Yaskawa INFORM job: A_ROOF_SIDE_0617_2_PAINT_1.JBI

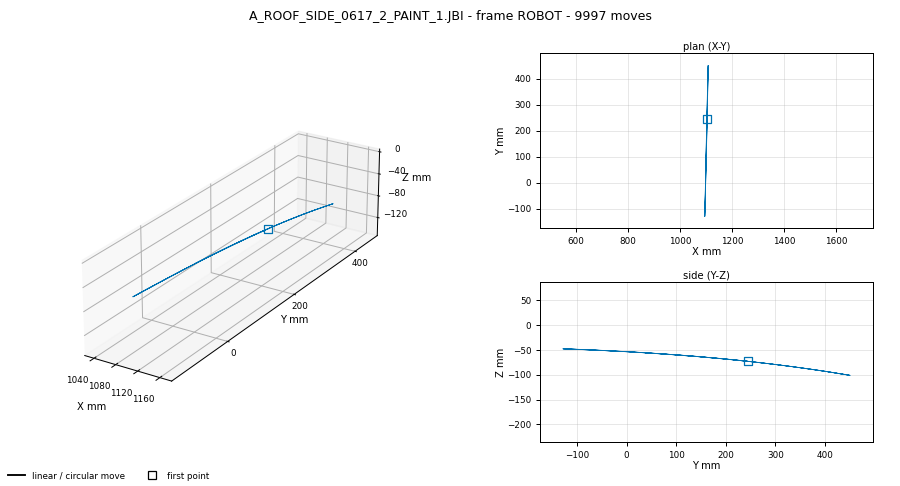
[picture p0: tool path of A_ROOF_SIDE_0617_2_PAINT_1.JBI in frame ROBOT, 9997 of 9997 moves have a stored position in this frame; points joined in program order, loops and branches not executed]
/JOB
//NAME A_ROOF_SIDE_0617_2_PAINT1
//POS
///NPOS 9997,0,0,0,0,0
///TOOL 1
///USER 0
///POSTYPE ROBOT
///RECTAN
///RCONF 1,0,0,0,0,0,0,0,0,0,0,0,0,0,0,0,0,0,0,0,0,0,0,0
C00000=1104.721,243.899,-72.511,179.198,14.617,151.233
C00001=1104.715,243.651,-72.485,179.194,14.617,151.234
C00002=1104.709,243.403,-72.458,179.190,14.617,151.234
C00003=1104.703,243.154,-72.431,179.186,14.617,151.235
C00004=1104.698,242.906,-72.404,179.183,14.617,151.236
C00005=1104.693,242.657,-72.378,179.179,14.617,151.237
C00006=1104.687,242.408,-72.352,179.175,14.617,151.238
C00007=1104.681,242.160,-72.325,179.171,14.616,151.238
C00008=1104.676,241.912,-72.298,179.167,14.617,151.239
C00009=1104.670,241.663,-72.272,179.163,14.616,151.240
C00010=1104.664,241.414,-72.246,179.159,14.616,151.241
C00011=1104.659,241.166,-72.219,179.155,14.616,151.242
C00012=1104.653,240.918,-72.192,179.151,14.616,151.243
C00013=1104.647,240.669,-72.166,179.148,14.616,151.244
C00014=1104.641,240.420,-72.140,179.144,14.616,151.244
C00015=1104.636,240.172,-72.113,179.140,14.616,151.245
C00016=1104.630,239.924,-72.086,179.136,14.616,151.246
C00017=1104.624,239.675,-72.060,179.132,14.616,151.247
C00018=1104.619,239.426,-72.034,179.129,14.616,151.248
C00019=1104.613,239.178,-72.007,179.125,14.616,151.249
C00020=1104.607,238.929,-71.981,179.121,14.616,151.250
C00021=1104.602,238.680,-71.955,179.117,14.616,151.250
C00022=1104.596,238.432,-71.928,179.113,14.616,151.251
C00023=1104.590,238.183,-71.902,179.110,14.616,151.252
C00024=1104.585,237.935,-71.875,179.105,14.615,151.253
C00025=1104.579,237.686,-71.849,179.101,14.615,151.254
C00026=1104.573,237.437,-71.823,179.097,14.615,151.254
C00027=1104.568,237.189,-71.796,179.094,14.615,151.255
C00028=1104.562,236.940,-71.770,179.090,14.615,151.256
C00029=1104.554,236.578,-71.732,179.084,14.615,151.257
C00030=1104.545,236.215,-71.694,179.078,14.615,151.259
C00031=1104.538,235.854,-71.656,179.073,14.615,151.260
C00032=1104.529,235.491,-71.618,179.067,14.615,151.261
C00033=1104.524,235.243,-71.591,179.063,14.615,151.262
C00034=1104.518,234.994,-71.565,179.059,14.615,151.263
C00035=1104.512,234.745,-71.538,179.056,14.615,151.264
C00036=1104.507,234.496,-71.513,179.052,14.615,151.264
C00037=1104.500,234.248,-71.486,179.048,14.615,151.265
C00038=1104.495,233.999,-71.461,179.044,14.615,151.266
C00039=1104.490,233.751,-71.435,179.040,14.615,151.267
C00040=1104.484,233.503,-71.408,179.037,14.615,151.268
C00041=1104.479,233.254,-71.382,179.033,14.615,151.269
C00042=1104.473,233.005,-71.357,179.029,14.615,151.270
C00043=1104.467,232.757,-71.330,179.025,14.615,151.270
C00044=1104.461,232.508,-71.304,179.021,14.615,151.271
C00045=1104.456,232.259,-71.279,179.017,14.615,151.272
C00046=1104.450,232.011,-71.253,179.014,14.615,151.273
C00047=1104.444,231.762,-71.227,179.010,14.615,151.274
C00048=1104.439,231.513,-71.201,179.006,14.615,151.275
C00049=1104.433,231.265,-71.174,179.002,14.615,151.276
C00050=1104.427,231.016,-71.149,178.998,14.615,151.276
C00051=1104.422,230.767,-71.123,178.994,14.615,151.277
C00052=1104.417,230.519,-71.098,178.991,14.616,151.278
C00053=1104.411,230.271,-71.071,178.987,14.616,151.279
C00054=1104.405,230.022,-71.046,178.983,14.615,151.280
C00055=1104.399,229.773,-71.020,178.979,14.615,151.281
C00056=1104.393,229.524,-70.994,178.975,14.616,151.282
C00057=1104.388,229.275,-70.968,178.972,14.616,151.282
C00058=1104.383,229.027,-70.943,178.968,14.616,151.283
C00059=1104.376,228.779,-70.917,178.964,14.616,151.284
C00060=1104.371,228.530,-70.891,178.960,14.616,151.285
C00061=1104.365,228.282,-70.865,178.956,14.616,151.286
C00062=1104.359,228.033,-70.840,178.952,14.616,151.287
C00063=1104.354,227.784,-70.814,178.948,14.616,151.288
C00064=1104.348,227.536,-70.789,178.944,14.616,151.289
C00065=1104.342,227.287,-70.763,178.941,14.617,151.290
C00066=1104.336,227.038,-70.737,178.937,14.617,151.290
C00067=1104.331,226.789,-70.711,178.933,14.616,151.291
C00068=1104.325,226.541,-70.686,178.929,14.616,151.292
C00069=1104.320,226.292,-70.661,178.925,14.617,151.293
C00070=1104.314,226.043,-70.635,178.921,14.617,151.294
C00071=1104.309,225.795,-70.610,178.918,14.617,151.295
C00072=1104.302,225.546,-70.584,178.914,14.617,151.296
C00073=1104.297,225.297,-70.558,178.910,14.617,151.296
C00074=1104.291,225.049,-70.533,178.906,14.617,151.297
C00075=1104.286,224.800,-70.507,178.902,14.617,151.298
C00076=1104.280,224.552,-70.482,178.898,14.617,151.299
C00077=1104.274,224.303,-70.456,178.894,14.617,151.300
C00078=1104.269,224.055,-70.431,178.891,14.617,151.301
C00079=1104.263,223.806,-70.405,178.887,14.617,151.302
C00080=1104.257,223.557,-70.380,178.883,14.617,151.302
C00081=1104.249,223.186,-70.342,178.877,14.618,151.304
C00082=1104.241,222.816,-70.304,178.871,14.618,151.305
C00083=1104.232,222.445,-70.267,178.866,14.618,151.306
C00084=1104.224,222.074,-70.228,178.860,14.619,151.308
C00085=1104.218,221.826,-70.203,178.857,14.619,151.309
C00086=1104.212,221.577,-70.179,178.853,14.619,151.310
C00087=1104.207,221.328,-70.153,178.849,14.619,151.310
C00088=1104.201,221.079,-70.127,178.845,14.619,151.311
C00089=1104.195,220.831,-70.102,178.841,14.619,151.312
C00090=1104.190,220.582,-70.077,178.837,14.620,151.313
C00091=1104.184,220.334,-70.052,178.833,14.620,151.314
C00092=1104.178,220.085,-70.027,178.829,14.620,151.315
C00093=1104.172,219.836,-70.002,178.826,14.620,151.316
C00094=1104.167,219.587,-69.977,178.822,14.620,151.317
C00095=1104.161,219.339,-69.951,178.818,14.620,151.317
C00096=1104.155,219.090,-69.926,178.814,14.620,151.318
C00097=1104.150,218.841,-69.901,178.810,14.620,151.319
C00098=1104.144,218.593,-69.876,178.806,14.620,151.320
C00099=1104.139,218.345,-69.851,178.803,14.620,151.321
C00100=1104.133,218.095,-69.826,178.799,14.620,151.322
C00101=1104.127,217.846,-69.800,178.796,14.621,151.323
C00102=1104.122,217.598,-69.776,178.792,14.621,151.324
C00103=1104.116,217.349,-69.751,178.788,14.621,151.324
C00104=1104.110,217.101,-69.726,178.784,14.622,151.325
C00105=1104.104,216.852,-69.701,178.780,14.622,151.326
C00106=1104.099,216.603,-69.676,178.776,14.622,151.327
C00107=1104.093,216.354,-69.651,178.772,14.622,151.328
C00108=1104.087,216.106,-69.626,178.768,14.622,151.329
C00109=1104.082,215.857,-69.601,178.764,14.622,151.330
C00110=1104.076,215.608,-69.576,178.761,14.622,151.331
C00111=1104.071,215.359,-69.551,178.757,14.623,151.332
C00112=1104.065,215.111,-69.526,178.753,14.623,151.332
C00113=1104.060,214.862,-69.502,178.749,14.623,151.333
C00114=1104.053,214.613,-69.476,178.745,14.623,151.334
C00115=1104.048,214.365,-69.452,178.742,14.624,151.335
C00116=1104.042,214.116,-69.427,178.738,14.624,151.336
C00117=1104.037,213.868,-69.402,178.734,14.624,151.337
C00118=1104.032,213.618,-69.377,178.730,14.624,151.338
C00119=1104.026,213.370,-69.352,178.726,14.624,151.339
C00120=1104.020,213.121,-69.328,178.723,14.624,151.340
C00121=1104.015,212.872,-69.303,178.719,14.625,151.340
C00122=1104.008,212.623,-69.278,178.715,14.625,151.341
C00123=1104.003,212.375,-69.254,178.711,14.625,151.342
C00124=1103.997,212.126,-69.229,178.707,14.625,151.343
C00125=1103.992,211.878,-69.204,178.703,14.625,151.344
C00126=1103.986,211.629,-69.180,178.699,14.625,151.345
C00127=1103.980,211.380,-69.155,178.696,14.626,151.346
C00128=1103.975,211.132,-69.130,178.692,14.626,151.347
C00129=1103.969,210.882,-69.106,178.688,14.626,151.348
C00130=1103.964,210.634,-69.081,178.684,14.627,151.348
C00131=1103.958,210.385,-69.057,178.681,14.627,151.349
C00132=1103.952,210.137,-69.032,178.677,14.627,151.350
C00133=1103.943,209.769,-68.996,178.671,14.628,151.352
C00134=1103.935,209.402,-68.960,178.666,14.628,151.353
C00135=1103.927,209.035,-68.923,178.660,14.628,151.354
C00136=1103.918,208.667,-68.887,178.654,14.628,151.356
C00137=1103.896,207.669,-68.790,178.625,14.626,151.361
C00138=1103.890,207.420,-68.765,178.621,14.626,151.362
C00139=1103.884,207.171,-68.741,178.617,14.628,151.364
C00140=1103.878,206.922,-68.717,178.613,14.628,151.365
C00141=1103.873,206.673,-68.692,178.609,14.630,151.366
C00142=1103.867,206.425,-68.669,178.605,14.631,151.367
C00143=1103.861,206.176,-68.644,178.600,14.632,151.368
C00144=1103.856,205.927,-68.620,178.597,14.633,151.369
C00145=1103.851,205.679,-68.596,178.592,14.634,151.370
C00146=1103.844,205.430,-68.572,178.589,14.635,151.372
C00147=1103.839,205.181,-68.547,178.584,14.636,151.373
C00148=1103.833,204.932,-68.523,178.580,14.637,151.374
C00149=1103.827,204.683,-68.498,178.576,14.638,151.375
C00150=1103.821,204.435,-68.475,178.572,14.639,151.376
C00151=1103.816,204.186,-68.450,178.568,14.640,151.377
C00152=1103.810,203.936,-68.427,178.564,14.641,151.378
C00153=1103.804,203.688,-68.403,178.560,14.642,151.379
C00154=1103.799,203.439,-68.379,178.556,14.643,151.381
C00155=1103.794,203.191,-68.354,178.552,14.644,151.382
C00156=1103.788,202.942,-68.330,178.547,14.645,151.383
C00157=1103.782,202.693,-68.306,178.544,14.646,151.384
C00158=1103.777,202.445,-68.282,178.539,14.647,151.385
C00159=1103.770,202.195,-68.259,178.536,14.648,151.386
C00160=1103.765,201.946,-68.234,178.531,14.649,151.387
C00161=1103.759,201.698,-68.211,178.527,14.650,151.388
C00162=1103.753,201.449,-68.186,178.524,14.651,151.389
C00163=1103.747,201.201,-68.162,178.519,14.652,151.391
C00164=1103.742,200.951,-68.139,178.516,14.654,151.392
C00165=1103.736,200.703,-68.115,178.511,14.655,151.393
C00166=1103.730,200.454,-68.091,178.508,14.656,151.394
C00167=1103.724,200.206,-68.067,178.503,14.657,151.395
C00168=1103.719,199.956,-68.043,178.499,14.658,151.396
C00169=1103.712,199.707,-68.019,178.495,14.659,151.397
C00170=1103.707,199.459,-67.995,178.491,14.660,151.399
C00171=1103.701,199.210,-67.972,178.487,14.661,151.400
C00172=1103.696,198.961,-67.948,178.483,14.662,151.401
C00173=1103.689,198.712,-67.924,178.479,14.663,151.402
C00174=1103.684,198.463,-67.900,178.475,14.664,151.403
C00175=1103.678,198.215,-67.877,178.471,14.665,151.404
C00176=1103.672,197.967,-67.853,178.467,14.666,151.405
C00177=1103.667,197.717,-67.829,178.463,14.667,151.406
C00178=1103.661,197.468,-67.805,178.459,14.668,151.407
C00179=1103.656,197.219,-67.782,178.455,14.669,151.409
C00180=1103.650,196.971,-67.758,178.451,14.670,151.410
C00181=1103.644,196.722,-67.734,178.447,14.671,151.411
C00182=1103.638,196.473,-67.711,178.443,14.672,151.412
C00183=1103.632,196.224,-67.687,178.439,14.672,151.413
C00184=1103.627,195.975,-67.663,178.435,14.674,151.414
C00185=1103.621,195.727,-67.640,178.431,14.675,151.415
C00186=1103.616,195.478,-67.616,178.427,14.676,151.416
C00187=1103.610,195.230,-67.593,178.423,14.677,151.417
C00188=1103.604,194.981,-67.570,178.419,14.677,151.418
C00189=1103.598,194.731,-67.545,178.415,14.679,151.420
C00190=1103.593,194.482,-67.522,178.411,14.680,151.421
C00191=1103.587,194.234,-67.498,178.407,14.681,151.422
C00192=1103.582,193.985,-67.475,178.403,14.681,151.423
C00193=1103.576,193.736,-67.452,178.399,14.682,151.424
C00194=1103.570,193.488,-67.428,178.396,14.683,151.425
C00195=1103.565,193.239,-67.405,178.391,14.684,151.426
C00196=1103.559,192.990,-67.381,178.387,14.686,151.427
C00197=1103.552,192.741,-67.358,178.383,14.686,151.428
C00198=1103.547,192.469,-67.332,178.379,14.687,151.429
C00199=1103.541,192.198,-67.307,178.375,14.688,151.431
C00200=1103.535,191.926,-67.281,178.371,14.690,151.432
C00201=1103.528,191.655,-67.255,178.366,14.690,151.433
C00202=1103.523,191.406,-67.232,178.362,14.691,151.434
C00203=1103.518,191.156,-67.209,178.358,14.693,151.435
C00204=1103.511,190.907,-67.185,178.354,14.693,151.436
C00205=1103.505,190.659,-67.162,178.350,14.694,151.437
C00206=1103.500,190.409,-67.138,178.347,14.695,151.438
C00207=1103.495,190.160,-67.115,178.342,14.696,151.439
C00208=1103.489,189.912,-67.092,178.339,14.697,151.440
C00209=1103.483,189.663,-67.069,178.335,14.698,151.442
C00210=1103.478,189.414,-67.045,178.330,14.699,151.443
C00211=1103.472,189.165,-67.022,178.327,14.700,151.444
C00212=1103.466,188.916,-66.999,178.323,14.700,151.445
C00213=1103.460,188.668,-66.976,178.319,14.702,151.446
C00214=1103.455,188.419,-66.952,178.315,14.702,151.447
C00215=1103.450,188.170,-66.929,178.312,14.704,151.448
C00216=1103.444,187.921,-66.906,178.307,14.704,151.449
C00217=1103.438,187.672,-66.883,178.303,14.705,151.450
C00218=1103.432,187.423,-66.860,178.300,14.706,151.451
C00219=1103.427,187.174,-66.837,178.296,14.706,151.452
C00220=1103.422,186.926,-66.814,178.292,14.708,151.453
C00221=1103.416,186.677,-66.791,178.288,14.708,151.454
C00222=1103.410,186.429,-66.768,178.284,14.709,151.455
C00223=1103.405,186.180,-66.745,178.280,14.710,151.456
C00224=1103.400,185.930,-66.721,178.276,14.711,151.457
C00225=1103.394,185.682,-66.698,178.273,14.712,151.458
C00226=1103.388,185.433,-66.675,178.269,14.713,151.459
C00227=1103.383,185.184,-66.652,178.265,14.713,151.460
C00228=1103.377,184.935,-66.629,178.261,14.714,151.461
C00229=1103.371,184.686,-66.607,178.257,14.716,151.463
C00230=1103.365,184.437,-66.584,178.253,14.717,151.464
C00231=1103.360,184.188,-66.561,178.249,14.718,151.465
C00232=1103.354,183.939,-66.538,178.245,14.719,151.466
C00233=1103.348,183.690,-66.515,178.241,14.719,151.467
C00234=1103.342,183.442,-66.492,178.237,14.720,151.468
C00235=1103.336,183.193,-66.469,178.234,14.721,151.469
C00236=1103.330,182.944,-66.446,178.230,14.722,151.470
C00237=1103.325,182.695,-66.424,178.226,14.723,151.471
C00238=1103.319,182.446,-66.401,178.222,14.724,151.472
C00239=1103.313,182.197,-66.378,178.219,14.725,151.473
C00240=1103.308,181.948,-66.355,178.214,14.726,151.474
C00241=1103.301,181.699,-66.333,178.211,14.727,151.475
C00242=1103.295,181.450,-66.310,178.207,14.728,151.476
C00243=1103.290,181.201,-66.287,178.202,14.728,151.477
C00244=1103.284,180.953,-66.264,178.199,14.730,151.478
C00245=1103.278,180.704,-66.241,178.195,14.730,151.479
C00246=1103.273,180.455,-66.218,178.191,14.732,151.481
C00247=1103.267,180.205,-66.196,178.187,14.732,151.481
C00248=1103.261,179.957,-66.174,178.184,14.733,151.482
C00249=1103.256,179.708,-66.151,178.180,14.734,151.484
C00250=1103.250,179.460,-66.128,178.175,14.734,151.485
C00251=1103.244,179.211,-66.105,178.172,14.736,151.486
C00252=1103.239,178.961,-66.083,178.168,14.736,151.487
C00253=1103.232,178.713,-66.061,178.165,14.737,151.488
C00254=1103.226,178.464,-66.038,178.160,14.738,151.489
C00255=1103.221,178.214,-66.016,178.157,14.739,151.490
C00256=1103.215,177.965,-65.993,178.153,14.740,151.491
C00257=1103.209,177.717,-65.971,178.149,14.741,151.492
C00258=1103.204,177.468,-65.948,178.145,14.742,151.493
C00259=1103.198,177.219,-65.925,178.141,14.742,151.494
C00260=1103.193,176.970,-65.902,178.138,14.744,151.495
C00261=1103.186,176.721,-65.880,178.133,14.744,151.496
C00262=1103.180,176.449,-65.856,178.129,14.745,151.497
C00263=1103.174,176.177,-65.831,178.126,14.746,151.498
C00264=1103.168,175.905,-65.807,178.122,14.747,151.499
C00265=1103.162,175.633,-65.782,178.117,14.748,151.500
C00266=1103.156,175.384,-65.760,178.113,14.748,151.501
C00267=1103.150,175.135,-65.737,178.110,14.750,151.502
C00268=1103.144,174.886,-65.715,178.106,14.750,151.503
C00269=1103.139,174.637,-65.692,178.102,14.751,151.504
C00270=1103.134,174.388,-65.670,178.098,14.752,151.505
C00271=1103.127,174.140,-65.648,178.095,14.753,151.506
C00272=1103.122,173.890,-65.626,178.091,14.753,151.507
C00273=1103.116,173.641,-65.603,178.086,14.754,151.509
C00274=1103.111,173.393,-65.581,178.083,14.755,151.509
C00275=1103.105,173.144,-65.559,178.079,14.756,151.510
C00276=1103.100,172.894,-65.536,178.076,14.757,151.511
C00277=1103.093,172.646,-65.514,178.072,14.757,151.512
C00278=1103.088,172.397,-65.492,178.068,14.759,151.513
C00279=1103.082,172.148,-65.469,178.064,14.759,151.514
C00280=1103.076,171.899,-65.448,178.061,14.760,151.515
C00281=1103.071,171.650,-65.425,178.057,14.760,151.516
C00282=1103.065,171.401,-65.403,178.053,14.761,151.517
C00283=1103.060,171.152,-65.381,178.050,14.762,151.518
C00284=1103.054,170.903,-65.358,178.045,14.763,151.519
C00285=1103.048,170.654,-65.337,178.042,14.764,151.520
C00286=1103.043,170.405,-65.314,178.038,14.764,151.521
C00287=1103.037,170.156,-65.292,178.035,14.765,151.522
C00288=1103.032,169.907,-65.270,178.031,14.766,151.523
C00289=1103.026,169.659,-65.247,178.027,14.766,151.524
C00290=1103.020,169.409,-65.226,178.023,14.767,151.525
C00291=1103.015,169.161,-65.204,178.019,14.768,151.526
C00292=1103.009,168.911,-65.182,178.016,14.769,151.527
C00293=1103.003,168.662,-65.159,178.012,14.769,151.528
C00294=1102.998,168.414,-65.138,178.009,14.770,151.529
C00295=1102.992,168.164,-65.116,178.005,14.771,151.530
C00296=1102.987,167.915,-65.094,178.002,14.772,151.531
C00297=1102.981,167.667,-65.072,177.997,14.772,151.532
C00298=1102.975,167.417,-65.049,177.993,14.773,151.533
C00299=1102.970,167.169,-65.028,177.990,14.774,151.534
C00300=1102.964,166.919,-65.006,177.986,14.774,151.535
C00301=1102.959,166.671,-64.983,177.983,14.775,151.536
C00302=1102.953,166.422,-64.962,177.979,14.776,151.537
C00303=1102.948,166.173,-64.940,177.976,14.777,151.538
C00304=1102.942,165.924,-64.918,177.972,14.777,151.539
C00305=1102.937,165.675,-64.896,177.969,14.778,151.540
C00306=1102.931,165.426,-64.875,177.964,14.779,151.541
C00307=1102.926,165.176,-64.853,177.960,14.779,151.542
C00308=1102.919,164.928,-64.830,177.957,14.780,151.542
C00309=1102.914,164.679,-64.808,177.953,14.780,151.543
C00310=1102.908,164.430,-64.787,177.950,14.782,151.544
C00311=1102.903,164.181,-64.765,177.946,14.782,151.545
C00312=1102.897,163.932,-64.743,177.943,14.783,151.546
C00313=1102.892,163.683,-64.721,177.939,14.783,151.547
C00314=1102.886,163.434,-64.700,177.935,14.784,151.548
C00315=1102.881,163.185,-64.678,177.932,14.785,151.549
C00316=1102.875,162.936,-64.656,177.928,14.785,151.550
C00317=1102.870,162.687,-64.635,177.925,14.786,151.551
C00318=1102.864,162.438,-64.613,177.921,14.786,151.552
C00319=1102.859,162.189,-64.591,177.917,14.787,151.553
C00320=1102.853,161.940,-64.569,177.913,14.788,151.554
C00321=1102.848,161.691,-64.548,177.910,14.789,151.555
C00322=1102.842,161.442,-64.526,177.906,14.789,151.556
C00323=1102.837,161.193,-64.504,177.902,14.789,151.557
C00324=1102.831,160.944,-64.483,177.899,14.791,151.558
C00325=1102.824,160.695,-64.461,177.895,14.791,151.559
C00326=1102.819,160.423,-64.437,177.892,14.792,151.560
C00327=1102.813,160.150,-64.415,177.888,14.792,151.560
C00328=1102.806,159.878,-64.391,177.883,14.793,151.562
C00329=1102.800,159.605,-64.367,177.879,14.794,151.563
C00330=1102.794,159.356,-64.346,177.876,14.795,151.564
C00331=1102.788,159.107,-64.324,177.872,14.795,151.564
C00332=1102.783,158.858,-64.302,177.869,14.796,151.565
C00333=1102.777,158.609,-64.281,177.865,14.797,151.566
C00334=1102.772,158.360,-64.260,177.862,14.798,151.567
C00335=1102.766,158.111,-64.238,177.858,14.798,151.568
C00336=1102.760,157.862,-64.217,177.854,14.798,151.569
C00337=1102.754,157.613,-64.195,177.851,14.799,151.570
C00338=1102.749,157.364,-64.174,177.847,14.799,151.571
C00339=1102.743,157.115,-64.153,177.844,14.800,151.572
C00340=1102.738,156.866,-64.131,177.840,14.801,151.573
C00341=1102.732,156.617,-64.110,177.836,14.802,151.574
C00342=1102.726,156.368,-64.089,177.832,14.802,151.575
C00343=1102.721,156.119,-64.068,177.829,14.803,151.576
C00344=1102.715,155.870,-64.046,177.825,14.804,151.577
C00345=1102.710,155.621,-64.024,177.822,14.804,151.577
C00346=1102.704,155.371,-64.004,177.818,14.805,151.578
C00347=1102.698,155.123,-63.982,177.815,14.806,151.579
C00348=1102.692,154.874,-63.961,177.811,14.806,151.580
C00349=1102.687,154.625,-63.939,177.807,14.806,151.581
C00350=1102.681,154.375,-63.918,177.804,14.807,151.582
C00351=1102.675,154.127,-63.897,177.800,14.807,151.583
C00352=1102.670,153.878,-63.877,177.797,14.808,151.584
C00353=1102.664,153.628,-63.855,177.793,14.809,151.585
C00354=1102.658,153.380,-63.834,177.790,14.810,151.586
C00355=1102.652,153.130,-63.813,177.786,14.810,151.586
C00356=1102.647,152.882,-63.792,177.783,14.811,151.587
C00357=1102.641,152.633,-63.770,177.779,14.811,151.588
C00358=1102.635,152.383,-63.749,177.776,14.812,151.589
C00359=1102.630,152.135,-63.728,177.772,14.812,151.590
C00360=1102.624,151.885,-63.707,177.769,14.813,151.591
C00361=1102.618,151.636,-63.686,177.765,14.814,151.592
C00362=1102.613,151.387,-63.665,177.761,14.814,151.593
C00363=1102.607,151.138,-63.644,177.758,14.815,151.594
C00364=1102.602,150.889,-63.623,177.754,14.815,151.595
C00365=1102.596,150.641,-63.602,177.751,14.816,151.596
C00366=1102.590,150.391,-63.581,177.747,14.816,151.596
C00367=1102.585,150.142,-63.560,177.744,14.817,151.597
C00368=1102.579,149.893,-63.539,177.740,14.817,151.598
C00369=1102.573,149.644,-63.517,177.737,14.818,151.599
C00370=1102.568,149.395,-63.497,177.733,14.818,151.600
C00371=1102.562,149.146,-63.476,177.730,14.819,151.601
C00372=1102.557,148.896,-63.455,177.726,14.820,151.602
C00373=1102.551,148.648,-63.433,177.723,14.821,151.603
C00374=1102.545,148.399,-63.414,177.719,14.821,151.603
C00375=1102.539,148.149,-63.393,177.717,14.821,151.604
C00376=1102.534,147.901,-63.371,177.713,14.822,151.605
C00377=1102.528,147.652,-63.351,177.710,14.823,151.606
C00378=1102.523,147.402,-63.330,177.706,14.823,151.607
C00379=1102.517,147.153,-63.309,177.702,14.823,151.608
C00380=1102.511,146.904,-63.289,177.699,14.824,151.609
C00381=1102.505,146.655,-63.267,177.695,14.825,151.610
C00382=1102.500,146.406,-63.246,177.692,14.825,151.610
C00383=1102.494,146.157,-63.226,177.688,14.825,151.611
C00384=1102.488,145.908,-63.206,177.685,14.826,151.612
C00385=1102.482,145.659,-63.184,177.681,14.827,151.613
C00386=1102.477,145.410,-63.164,177.678,14.828,151.614
C00387=1102.472,145.161,-63.143,177.674,14.827,151.615
C00388=1102.465,144.912,-63.122,177.671,14.828,151.616
C00389=1102.459,144.663,-63.102,177.667,14.829,151.617
C00390=1102.453,144.390,-63.079,177.663,14.829,151.618
C00391=1102.447,144.117,-63.056,177.660,14.830,151.618
C00392=1102.441,143.845,-63.034,177.656,14.830,151.619
C00393=1102.435,143.572,-63.011,177.652,14.831,151.620
C00394=1102.429,143.322,-62.990,177.649,14.832,151.621
C00395=1102.424,143.073,-62.970,177.645,14.832,151.622
C00396=1102.418,142.824,-62.950,177.642,14.832,151.623
C00397=1102.413,142.575,-62.929,177.639,14.833,151.624
C00398=1102.407,142.327,-62.908,177.635,14.834,151.625
C00399=1102.401,142.077,-62.887,177.632,14.833,151.625
C00400=1102.395,141.828,-62.867,177.629,14.834,151.626
C00401=1102.390,141.579,-62.846,177.625,14.835,151.627
C00402=1102.385,141.330,-62.826,177.622,14.835,151.628
C00403=1102.379,141.081,-62.806,177.618,14.836,151.629
C00404=1102.373,140.831,-62.785,177.614,14.835,151.630
C00405=1102.368,140.582,-62.764,177.611,14.836,151.630
C00406=1102.362,140.333,-62.744,177.607,14.837,151.631
C00407=1102.356,140.084,-62.724,177.605,14.837,151.632
C00408=1102.350,139.835,-62.704,177.601,14.838,151.633
C00409=1102.344,139.586,-62.683,177.598,14.838,151.634
C00410=1102.339,139.337,-62.662,177.594,14.838,151.635
C00411=1102.333,139.088,-62.642,177.591,14.839,151.636
C00412=1102.328,138.839,-62.621,177.587,14.839,151.636
C00413=1102.322,138.590,-62.601,177.584,14.840,151.637
C00414=1102.316,138.341,-62.581,177.581,14.840,151.638
C00415=1102.310,138.091,-62.561,177.577,14.841,151.639
C00416=1102.305,137.842,-62.541,177.574,14.841,151.640
C00417=1102.300,137.593,-62.520,177.571,14.842,151.640
C00418=1102.294,137.344,-62.500,177.567,14.842,151.641
C00419=1102.288,137.095,-62.480,177.564,14.843,151.642
C00420=1102.282,136.846,-62.460,177.560,14.843,151.643
C00421=1102.277,136.597,-62.439,177.557,14.844,151.644
C00422=1102.271,136.347,-62.419,177.554,14.843,151.645
C00423=1102.265,136.098,-62.398,177.550,14.844,151.645
C00424=1102.259,135.850,-62.378,177.547,14.844,151.646
C00425=1102.253,135.601,-62.358,177.544,14.845,151.647
C00426=1102.248,135.352,-62.338,177.540,14.845,151.648
C00427=1102.242,135.102,-62.318,177.537,14.846,151.649
C00428=1102.237,134.853,-62.298,177.533,14.846,151.649
C00429=1102.231,134.604,-62.278,177.530,14.847,151.650
C00430=1102.226,134.355,-62.257,177.527,14.847,151.651
C00431=1102.220,134.106,-62.237,177.524,14.847,151.652
C00432=1102.214,133.856,-62.216,177.520,14.848,151.653
C00433=1102.208,133.607,-62.197,177.517,14.848,151.654
C00434=1102.203,133.358,-62.177,177.513,14.849,151.654
C00435=1102.197,133.109,-62.157,177.510,14.849,151.655
C00436=1102.191,132.860,-62.137,177.507,14.849,151.656
C00437=1102.186,132.611,-62.117,177.504,14.850,151.657
C00438=1102.180,132.362,-62.097,177.500,14.850,151.658
C00439=1102.175,132.113,-62.076,177.497,14.850,151.658
C00440=1102.169,131.864,-62.056,177.493,14.851,151.659
C00441=1102.163,131.614,-62.037,177.491,14.851,151.660
C00442=1102.157,131.366,-62.017,177.487,14.851,151.661
C00443=1102.152,131.116,-61.997,177.484,14.852,151.662
C00444=1102.146,130.867,-61.977,177.480,14.852,151.662
C00445=1102.140,130.618,-61.957,177.477,14.853,151.663
C00446=1102.134,130.369,-61.938,177.474,14.853,151.664
C00447=1102.129,130.119,-61.917,177.471,14.853,151.665
C00448=1102.123,129.870,-61.897,177.467,14.854,151.666
C00449=1102.117,129.621,-61.877,177.464,14.854,151.666
C00450=1102.111,129.372,-61.858,177.460,14.854,151.667
C00451=1102.106,129.123,-61.838,177.457,14.855,151.668
C00452=1102.100,128.873,-61.818,177.454,14.855,151.669
C00453=1102.094,128.625,-61.798,177.451,14.856,151.670
C00454=1102.088,128.352,-61.777,177.447,14.856,151.670
C00455=1102.081,128.079,-61.754,177.443,14.856,151.671
C00456=1102.075,127.807,-61.734,177.440,14.856,151.672
C00457=1102.070,127.533,-61.712,177.436,14.857,151.673
C00458=1102.064,127.284,-61.692,177.433,14.857,151.674
C00459=1102.058,127.035,-61.672,177.430,14.858,151.675
C00460=1102.052,126.786,-61.653,177.426,14.857,151.675
C00461=1102.046,126.537,-61.633,177.423,14.858,151.676
C00462=1102.041,126.288,-61.614,177.420,14.858,151.677
C00463=1102.035,126.038,-61.593,177.417,14.859,151.678
C00464=1102.030,125.789,-61.574,177.413,14.859,151.678
C00465=1102.024,125.540,-61.554,177.410,14.859,151.679
C00466=1102.018,125.291,-61.535,177.407,14.859,151.680
C00467=1102.012,125.042,-61.515,177.404,14.860,151.681
C00468=1102.006,124.793,-61.496,177.400,14.860,151.682
C00469=1102.000,124.544,-61.476,177.397,14.861,151.682
C00470=1101.995,124.294,-61.456,177.394,14.861,151.683
C00471=1101.990,124.045,-61.437,177.391,14.861,151.684
C00472=1101.984,123.796,-61.417,177.387,14.861,151.685
C00473=1101.978,123.546,-61.398,177.384,14.862,151.685
C00474=1101.972,123.297,-61.378,177.381,14.861,151.686
C00475=1101.967,123.049,-61.359,177.378,14.862,151.687
C00476=1101.961,122.799,-61.339,177.375,14.862,151.688
C00477=1101.955,122.550,-61.320,177.372,14.862,151.688
C00478=1101.950,122.301,-61.300,177.368,14.863,151.689
C00479=1101.945,122.051,-61.280,177.365,14.863,151.690
C00480=1101.939,121.803,-61.260,177.361,14.863,151.691
C00481=1101.933,121.553,-61.241,177.359,14.864,151.691
C00482=1101.927,121.304,-61.222,177.355,14.864,151.692
C00483=1101.922,121.055,-61.203,177.352,14.864,151.693
C00484=1101.916,120.806,-61.183,177.349,14.864,151.694
C00485=1101.910,120.557,-61.164,177.346,14.864,151.694
C00486=1101.905,120.307,-61.145,177.343,14.865,151.695
C00487=1101.899,120.058,-61.125,177.340,14.865,151.696
C00488=1101.893,119.809,-61.105,177.337,14.865,151.696
C00489=1101.888,119.560,-61.087,177.333,14.865,151.697
C00490=1101.882,119.311,-61.067,177.330,14.866,151.698
C00491=1101.877,119.061,-61.048,177.327,14.866,151.699
C00492=1101.871,118.812,-61.029,177.324,14.866,151.699
C00493=1101.865,118.563,-61.009,177.320,14.866,151.700
C00494=1101.860,118.314,-60.990,177.318,14.867,151.701
C00495=1101.854,118.065,-60.971,177.314,14.866,151.702
C00496=1101.848,117.816,-60.952,177.312,14.867,151.702
C00497=1101.843,117.566,-60.932,177.308,14.866,151.703
C00498=1101.837,117.317,-60.913,177.305,14.867,151.704
C00499=1101.832,117.068,-60.894,177.302,14.867,151.705
C00500=1101.826,116.819,-60.874,177.299,14.867,151.705
C00501=1101.820,116.570,-60.855,177.295,14.867,151.706
C00502=1101.815,116.320,-60.836,177.293,14.867,151.707
C00503=1101.810,116.072,-60.817,177.289,14.867,151.707
C00504=1101.804,115.822,-60.798,177.286,14.868,151.708
C00505=1101.798,115.573,-60.778,177.283,14.868,151.709
C00506=1101.792,115.323,-60.759,177.280,14.868,151.710
C00507=1101.787,115.075,-60.740,177.277,14.868,151.710
C00508=1101.782,114.825,-60.721,177.274,14.868,151.711
C00509=1101.776,114.576,-60.702,177.270,14.868,151.712
C00510=1101.771,114.327,-60.683,177.267,14.869,151.712
C00511=1101.764,114.078,-60.664,177.264,14.868,151.713
C00512=1101.759,113.828,-60.645,177.261,14.869,151.714
C00513=1101.753,113.579,-60.626,177.258,14.869,151.714
C00514=1101.748,113.330,-60.607,177.255,14.869,151.715
C00515=1101.742,113.081,-60.588,177.252,14.869,151.716
C00516=1101.736,112.832,-60.569,177.249,14.869,151.717
C00517=1101.730,112.582,-60.550,177.246,14.870,151.717
C00518=1101.725,112.309,-60.530,177.242,14.870,151.718
C00519=1101.718,112.036,-60.508,177.239,14.870,151.719
C00520=1101.712,111.764,-60.488,177.235,14.870,151.720
C00521=1101.706,111.491,-60.467,177.232,14.870,151.720
C00522=1101.700,111.241,-60.447,177.229,14.870,151.721
C00523=1101.694,110.993,-60.429,177.226,14.871,151.722
C00524=1101.689,110.743,-60.411,177.223,14.870,151.722
C00525=1101.683,110.493,-60.391,177.220,14.871,151.723
C00526=1101.677,110.244,-60.373,177.216,14.871,151.724
C00527=1101.672,109.995,-60.354,177.213,14.871,151.725
C00528=1101.666,109.746,-60.335,177.210,14.871,151.725
C00529=1101.660,109.497,-60.316,177.207,14.871,151.726
C00530=1101.655,109.248,-60.297,177.205,14.872,151.727
C00531=1101.649,108.998,-60.279,177.201,14.871,151.727
C00532=1101.643,108.749,-60.260,177.198,14.872,151.728
C00533=1101.638,108.500,-60.241,177.195,14.872,151.729
C00534=1101.632,108.251,-60.222,177.192,14.872,151.729
C00535=1101.626,108.001,-60.204,177.189,14.872,151.730
C00536=1101.621,107.752,-60.185,177.186,14.872,151.731
C00537=1101.615,107.503,-60.166,177.183,14.872,151.731
C00538=1101.609,107.254,-60.147,177.180,14.872,151.732
C00539=1101.604,107.004,-60.129,177.177,14.872,151.733
C00540=1101.597,106.755,-60.110,177.174,14.872,151.733
C00541=1101.592,106.506,-60.091,177.170,14.872,151.734
C00542=1101.587,106.257,-60.072,177.168,14.873,151.735
C00543=1101.581,106.007,-60.054,177.165,14.873,151.735
C00544=1101.575,105.758,-60.035,177.162,14.873,151.736
C00545=1101.569,105.510,-60.017,177.159,14.873,151.737
C00546=1101.564,105.260,-59.998,177.155,14.873,151.737
C00547=1101.558,105.011,-59.980,177.153,14.873,151.738
C00548=1101.552,104.761,-59.961,177.149,14.873,151.739
C00549=1101.547,104.512,-59.942,177.147,14.873,151.739
C00550=1101.541,104.263,-59.924,177.143,14.873,151.740
C00551=1101.536,104.013,-59.905,177.141,14.873,151.741
C00552=1101.530,103.765,-59.887,177.137,14.873,151.741
C00553=1101.524,103.515,-59.869,177.135,14.873,151.742
C00554=1101.518,103.266,-59.850,177.131,14.873,151.743
C00555=1101.513,103.017,-59.831,177.129,14.873,151.743
C00556=1101.507,102.767,-59.813,177.126,14.873,151.744
C00557=1101.502,102.518,-59.794,177.123,14.873,151.745
C00558=1101.496,102.268,-59.776,177.120,14.873,151.745
C00559=1101.490,102.020,-59.757,177.116,14.873,151.746
C00560=1101.485,101.770,-59.739,177.114,14.873,151.747
C00561=1101.479,101.521,-59.721,177.110,14.873,151.747
C00562=1101.474,101.271,-59.702,177.108,14.873,151.748
C00563=1101.468,101.023,-59.684,177.105,14.873,151.749
C00564=1101.462,100.773,-59.666,177.102,14.873,151.749
C00565=1101.457,100.524,-59.647,177.098,14.873,151.750
C00566=1101.451,100.275,-59.629,177.096,14.873,151.751
C00567=1101.445,100.025,-59.610,177.093,14.873,151.751
C00568=1101.439,99.776,-59.592,177.090,14.873,151.752
C00569=1101.433,99.527,-59.574,177.087,14.873,151.753
C00570=1101.428,99.278,-59.555,177.084,14.873,151.753
C00571=1101.422,99.028,-59.537,177.081,14.873,151.754
C00572=1101.416,98.780,-59.519,177.078,14.873,151.754
C00573=1101.411,98.530,-59.501,177.075,14.873,151.755
C00574=1101.405,98.281,-59.482,177.072,14.873,151.756
C00575=1101.399,98.031,-59.464,177.069,14.873,151.756
C00576=1101.394,97.782,-59.446,177.067,14.873,151.757
C00577=1101.388,97.533,-59.428,177.063,14.873,151.758
C00578=1101.382,97.284,-59.410,177.060,14.873,151.758
C00579=1101.377,97.034,-59.392,177.057,14.873,151.759
C00580=1101.371,96.785,-59.373,177.054,14.873,151.760
C00581=1101.365,96.536,-59.355,177.051,14.873,151.760
C00582=1101.359,96.263,-59.335,177.049,14.873,151.761
C00583=1101.353,95.990,-59.315,177.045,14.873,151.762
C00584=1101.346,95.718,-59.296,177.042,14.872,151.762
C00585=1101.340,95.444,-59.275,177.039,14.873,151.763
C00586=1101.335,95.195,-59.258,177.036,14.872,151.764
C00587=1101.329,94.945,-59.240,177.033,14.873,151.764
C00588=1101.324,94.696,-59.222,177.030,14.873,151.765
C00589=1101.318,94.448,-59.203,177.027,14.873,151.765
C00590=1101.312,94.198,-59.185,177.025,14.873,151.766
C00591=1101.306,93.949,-59.168,177.021,14.872,151.767
C00592=1101.301,93.699,-59.149,177.019,14.872,151.767
C00593=1101.295,93.450,-59.132,177.015,14.872,151.768
C00594=1101.289,93.201,-59.113,177.013,14.872,151.768
C00595=1101.283,92.952,-59.095,177.009,14.872,151.769
C00596=1101.279,92.702,-59.077,177.007,14.872,151.770
C00597=1101.273,92.453,-59.059,177.004,14.872,151.770
C00598=1101.267,92.203,-59.042,177.001,14.872,151.771
C00599=1101.261,91.954,-59.024,176.999,14.872,151.771
C00600=1101.255,91.705,-59.006,176.995,14.871,151.772
C00601=1101.250,91.456,-58.987,176.993,14.872,151.773
C00602=1101.244,91.206,-58.970,176.989,14.871,151.773
C00603=1101.239,90.957,-58.952,176.987,14.871,151.774
C00604=1101.233,90.708,-58.934,176.983,14.871,151.775
C00605=1101.227,90.458,-58.916,176.981,14.871,151.775
C00606=1101.222,90.209,-58.899,176.978,14.871,151.776
C00607=1101.215,89.960,-58.881,176.975,14.871,151.776
C00608=1101.210,89.711,-58.863,176.973,14.871,151.777
C00609=1101.204,89.462,-58.846,176.969,14.870,151.777
C00610=1101.199,89.211,-58.827,176.967,14.871,151.778
C00611=1101.193,88.962,-58.810,176.963,14.870,151.779
C00612=1101.187,88.713,-58.792,176.961,14.871,151.779
C00613=1101.182,88.464,-58.774,176.958,14.871,151.780
C00614=1101.176,88.215,-58.756,176.955,14.870,151.781
C00615=1101.170,87.966,-58.738,176.953,14.870,151.781
C00616=1101.164,87.716,-58.720,176.949,14.870,151.782
C00617=1101.159,87.467,-58.703,176.947,14.870,151.782
C00618=1101.153,87.217,-58.686,176.944,14.869,151.783
C00619=1101.148,86.968,-58.668,176.941,14.870,151.783
C00620=1101.141,86.718,-58.650,176.938,14.870,151.784
C00621=1101.136,86.469,-58.633,176.935,14.869,151.785
C00622=1101.130,86.220,-58.615,176.933,14.869,151.785
C00623=1101.125,85.971,-58.597,176.929,14.869,151.786
C00624=1101.119,85.721,-58.580,176.927,14.869,151.786
C00625=1101.113,85.472,-58.562,176.924,14.869,151.787
C00626=1101.108,85.223,-58.544,176.921,14.869,151.788
C00627=1101.102,84.974,-58.526,176.919,14.869,151.788
C00628=1101.096,84.725,-58.509,176.915,14.868,151.789
C00629=1101.091,84.476,-58.491,176.913,14.868,151.789
C00630=1101.085,84.225,-58.474,176.910,14.868,151.790
C00631=1101.079,83.976,-58.457,176.907,14.868,151.790
C00632=1101.074,83.727,-58.439,176.905,14.868,151.791
C00633=1101.067,83.478,-58.422,176.902,14.867,151.791
C00634=1101.061,83.229,-58.404,176.899,14.867,151.792
C00635=1101.056,82.980,-58.386,176.896,14.867,151.793
C00636=1101.051,82.730,-58.370,176.893,14.867,151.793
C00637=1101.045,82.481,-58.352,176.891,14.867,151.794
C00638=1101.039,82.231,-58.334,176.888,14.866,151.794
C00639=1101.033,81.982,-58.317,176.885,14.867,151.795
C00640=1101.028,81.732,-58.300,176.882,14.866,151.795
C00641=1101.023,81.483,-58.282,176.880,14.866,151.796
C00642=1101.017,81.234,-58.264,176.876,14.865,151.797
C00643=1101.011,80.985,-58.247,176.874,14.865,151.797
C00644=1101.006,80.735,-58.230,176.871,14.866,151.798
C00645=1101.000,80.486,-58.212,176.868,14.865,151.798
C00646=1100.993,80.213,-58.194,176.866,14.865,151.799
C00647=1100.987,79.941,-58.174,176.862,14.865,151.800
C00648=1100.981,79.667,-58.155,176.859,14.864,151.800
C00649=1100.975,79.394,-58.136,176.857,14.864,151.801
C00650=1100.969,79.145,-58.119,176.854,14.863,151.801
C00651=1100.964,78.896,-58.102,176.851,14.864,151.802
C00652=1100.959,78.646,-58.084,176.848,14.863,151.802
C00653=1100.952,78.398,-58.068,176.845,14.863,151.803
C00654=1100.947,78.147,-58.050,176.843,14.863,151.803
C00655=1100.941,77.898,-58.033,176.840,14.862,151.804
C00656=1100.936,77.649,-58.015,176.837,14.862,151.805
C00657=1100.930,77.400,-57.999,176.834,14.862,151.805
C00658=1100.924,77.151,-57.981,176.832,14.862,151.806
C00659=1100.918,76.901,-57.964,176.829,14.862,151.806
C00660=1100.913,76.652,-57.947,176.826,14.861,151.807
C00661=1100.907,76.403,-57.930,176.824,14.861,151.807
C00662=1100.901,76.153,-57.913,176.821,14.861,151.808
C00663=1100.896,75.904,-57.895,176.818,14.861,151.808
C00664=1100.890,75.655,-57.879,176.816,14.861,151.809
C00665=1100.884,75.405,-57.861,176.812,14.860,151.809
C00666=1100.879,75.155,-57.844,176.810,14.860,151.810
C00667=1100.872,74.907,-57.827,176.808,14.860,151.810
C00668=1100.867,74.657,-57.810,176.804,14.860,151.811
C00669=1100.862,74.408,-57.793,176.802,14.859,151.811
C00670=1100.856,74.159,-57.776,176.799,14.859,151.812
C00671=1100.849,73.909,-57.759,176.796,14.859,151.813
C00672=1100.844,73.659,-57.742,176.794,14.859,151.813
C00673=1100.838,73.410,-57.725,176.791,14.858,151.814
C00674=1100.833,73.161,-57.708,176.788,14.858,151.814
C00675=1100.827,72.912,-57.690,176.785,14.857,151.815
C00676=1100.821,72.662,-57.674,176.783,14.857,151.815
C00677=1100.816,72.413,-57.657,176.781,14.857,151.816
C00678=1100.811,72.164,-57.640,176.777,14.857,151.816
C00679=1100.805,71.914,-57.623,176.775,14.857,151.817
C00680=1100.798,71.665,-57.605,176.772,14.856,151.817
C00681=1100.793,71.415,-57.589,176.770,14.856,151.818
C00682=1100.787,71.166,-57.572,176.767,14.856,151.818
C00683=1100.782,70.917,-57.555,176.764,14.855,151.819
C00684=1100.776,70.667,-57.539,176.762,14.855,151.819
C00685=1100.770,70.418,-57.521,176.759,14.855,151.820
C00686=1100.764,70.169,-57.505,176.756,14.855,151.820
C00687=1100.759,69.919,-57.488,176.754,14.854,151.821
C00688=1100.754,69.670,-57.470,176.751,14.854,151.822
C00689=1100.748,69.421,-57.454,176.748,14.853,151.822
C00690=1100.742,69.171,-57.437,176.746,14.854,151.822
C00691=1100.737,68.922,-57.421,176.743,14.853,151.823
C00692=1100.731,68.673,-57.403,176.740,14.853,151.824
C00693=1100.724,68.423,-57.387,176.738,14.852,151.824
C00694=1100.719,68.173,-57.370,176.735,14.852,151.825
C00695=1100.713,67.924,-57.353,176.733,14.852,151.825
C00696=1100.708,67.675,-57.336,176.730,14.851,151.826
C00697=1100.702,67.425,-57.320,176.727,14.851,151.826
C00698=1100.696,67.176,-57.304,176.725,14.851,151.827
C00699=1100.690,66.927,-57.286,176.722,14.850,151.827
C00700=1100.684,66.678,-57.270,176.719,14.850,151.828
C00701=1100.679,66.428,-57.253,176.716,14.849,151.828
C00702=1100.673,66.179,-57.237,176.714,14.849,151.829
C00703=1100.668,65.929,-57.220,176.712,14.849,151.829
C00704=1100.662,65.680,-57.203,176.708,14.849,151.830
C00705=1100.657,65.430,-57.186,176.706,14.848,151.830
C00706=1100.651,65.181,-57.170,176.704,14.848,151.830
C00707=1100.645,64.932,-57.153,176.701,14.847,151.831
C00708=1100.639,64.682,-57.137,176.699,14.847,151.831
C00709=1100.634,64.433,-57.120,176.696,14.847,151.832
C00710=1100.627,64.160,-57.102,176.693,14.846,151.832
C00711=1100.621,63.887,-57.083,176.690,14.846,151.833
C00712=1100.615,63.614,-57.066,176.687,14.846,151.834
C00713=1100.608,63.341,-57.048,176.684,14.846,151.834
C00714=1100.602,63.092,-57.031,176.682,14.845,151.835
C00715=1100.597,62.842,-57.014,176.679,14.844,151.835
C00716=1100.591,62.593,-56.998,176.676,14.844,151.836
C00717=1100.585,62.343,-56.982,176.674,14.844,151.836
C00718=1100.579,62.094,-56.966,176.671,14.844,151.837
C00719=1100.574,61.844,-56.949,176.669,14.843,151.837
C00720=1100.568,61.595,-56.933,176.666,14.843,151.838
C00721=1100.562,61.346,-56.916,176.663,14.843,151.838
C00722=1100.555,61.097,-56.899,176.661,14.842,151.839
C00723=1100.550,60.848,-56.883,176.659,14.842,151.839
C00724=1100.544,60.598,-56.866,176.656,14.841,151.840
C00725=1100.538,60.349,-56.850,176.653,14.841,151.840
C00726=1100.532,60.099,-56.834,176.651,14.841,151.841
C00727=1100.526,59.850,-56.817,176.648,14.840,151.841
C00728=1100.521,59.601,-56.801,176.646,14.840,151.842
C00729=1100.516,59.350,-56.785,176.643,14.840,151.842
C00730=1100.510,59.101,-56.769,176.640,14.839,151.842
C00731=1100.504,58.852,-56.753,176.638,14.839,151.843
C00732=1100.498,58.603,-56.737,176.636,14.839,151.843
C00733=1100.492,58.354,-56.720,176.633,14.838,151.844
C00734=1100.487,58.104,-56.704,176.631,14.838,151.844
C00735=1100.481,57.855,-56.687,176.627,14.837,151.845
C00736=1100.475,57.605,-56.671,176.625,14.837,151.845
C00737=1100.469,57.356,-56.655,176.623,14.837,151.846
C00738=1100.463,57.107,-56.639,176.620,14.836,151.846
C00739=1100.457,56.857,-56.622,176.617,14.836,151.847
C00740=1100.452,56.608,-56.605,176.615,14.836,151.847
C00741=1100.447,56.358,-56.590,176.612,14.835,151.848
C00742=1100.441,56.108,-56.574,176.610,14.835,151.848
C00743=1100.435,55.860,-56.558,176.608,14.835,151.849
C00744=1100.429,55.610,-56.541,176.605,14.834,151.849
C00745=1100.423,55.361,-56.525,176.602,14.833,151.849
C00746=1100.417,55.112,-56.509,176.600,14.833,151.850
C00747=1100.412,54.862,-56.493,176.597,14.833,151.850
C00748=1100.407,54.612,-56.477,176.595,14.832,151.851
C00749=1100.401,54.363,-56.460,176.593,14.832,151.851
C00750=1100.395,54.114,-56.444,176.590,14.831,151.852
C00751=1100.390,53.864,-56.429,176.587,14.831,151.852
C00752=1100.384,53.615,-56.413,176.585,14.831,151.853
C00753=1100.378,53.365,-56.396,176.582,14.830,151.853
C00754=1100.372,53.116,-56.380,176.580,14.830,151.854
C00755=1100.366,52.866,-56.365,176.578,14.829,151.854
C00756=1100.361,52.617,-56.349,176.575,14.828,151.854
C00757=1100.355,52.368,-56.332,176.572,14.828,151.855
C00758=1100.350,52.118,-56.316,176.570,14.828,151.855
C00759=1100.344,51.868,-56.300,176.567,14.827,151.856
C00760=1100.338,51.619,-56.284,176.565,14.827,151.856
C00761=1100.333,51.370,-56.268,176.563,14.827,151.857
C00762=1100.327,51.120,-56.252,176.560,14.826,151.857
C00763=1100.321,50.871,-56.236,176.557,14.825,151.858
C00764=1100.315,50.622,-56.220,176.555,14.825,151.858
C00765=1100.309,50.372,-56.204,176.552,14.824,151.858
C00766=1100.304,50.123,-56.188,176.550,14.824,151.859
C00767=1100.298,49.874,-56.172,176.548,14.824,151.859
C00768=1100.293,49.624,-56.157,176.545,14.823,151.860
C00769=1100.287,49.374,-56.140,176.543,14.822,151.860
C00770=1100.282,49.125,-56.125,176.541,14.822,151.861
C00771=1100.276,48.876,-56.109,176.538,14.821,151.861
C00772=1100.270,48.626,-56.093,176.535,14.821,151.861
C00773=1100.264,48.376,-56.077,176.533,14.820,151.862
C00774=1100.258,48.104,-56.060,176.530,14.820,151.862
C00775=1100.252,47.830,-56.042,176.528,14.820,151.863
C00776=1100.246,47.558,-56.025,176.525,14.819,151.863
C00777=1100.239,47.284,-56.007,176.522,14.818,151.864
C00778=1100.234,47.035,-55.992,176.520,14.817,151.864
C00779=1100.228,46.785,-55.976,176.517,14.817,151.865
C00780=1100.222,46.535,-55.960,176.515,14.817,151.865
C00781=1100.217,46.287,-55.945,176.512,14.816,151.865
C00782=1100.211,46.037,-55.929,176.510,14.816,151.866
C00783=1100.206,45.787,-55.913,176.508,14.815,151.866
C00784=1100.200,45.538,-55.898,176.505,14.814,151.867
C00785=1100.195,45.289,-55.881,176.503,14.814,151.867
C00786=1100.189,45.039,-55.866,176.501,14.814,151.868
C00787=1100.184,44.790,-55.850,176.498,14.813,151.868
C00788=1100.178,44.540,-55.834,176.495,14.813,151.868
C00789=1100.172,44.290,-55.819,176.494,14.812,151.869
C00790=1100.167,44.042,-55.803,176.491,14.811,151.869
C00791=1100.161,43.792,-55.787,176.488,14.811,151.870
C00792=1100.155,43.543,-55.772,176.486,14.810,151.870
C00793=1100.150,43.293,-55.757,176.483,14.809,151.870
C00794=1100.144,43.043,-55.741,176.481,14.809,151.871
C00795=1100.138,42.794,-55.725,176.479,14.809,151.871
C00796=1100.133,42.545,-55.710,176.476,14.808,151.872
C00797=1100.126,42.296,-55.694,176.474,14.807,151.872
C00798=1100.121,42.046,-55.678,176.472,14.807,151.873
C00799=1100.116,41.797,-55.663,176.469,14.807,151.873
C00800=1100.110,41.547,-55.647,176.466,14.806,151.873
C00801=1100.104,41.297,-55.631,176.464,14.806,151.874
C00802=1100.098,41.048,-55.617,176.462,14.805,151.874
C00803=1100.092,40.799,-55.601,176.459,14.804,151.875
C00804=1100.087,40.549,-55.585,176.457,14.804,151.875
C00805=1100.081,40.300,-55.570,176.455,14.803,151.875
C00806=1100.075,40.051,-55.554,176.452,14.802,151.876
C00807=1100.069,39.801,-55.539,176.450,14.802,151.876
C00808=1100.064,39.551,-55.523,176.448,14.802,151.877
C00809=1100.058,39.301,-55.508,176.445,14.802,151.877
C00810=1100.052,39.052,-55.492,176.443,14.800,151.877
C00811=1100.047,38.803,-55.477,176.441,14.800,151.878
C00812=1100.041,38.553,-55.462,176.438,14.800,151.878
C00813=1100.036,38.304,-55.446,176.435,14.799,151.879
C00814=1100.029,38.055,-55.431,176.433,14.798,151.879
C00815=1100.024,37.805,-55.415,176.431,14.798,151.879
C00816=1100.019,37.556,-55.400,176.429,14.797,151.880
C00817=1100.012,37.306,-55.385,176.426,14.796,151.880
C00818=1100.007,37.057,-55.370,176.424,14.796,151.881
C00819=1100.001,36.808,-55.354,176.422,14.796,151.881
C00820=1099.995,36.558,-55.339,176.419,14.795,151.881
C00821=1099.990,36.308,-55.324,176.417,14.794,151.882
C00822=1099.983,36.059,-55.309,176.415,14.794,151.882
C00823=1099.978,35.809,-55.293,176.413,14.793,151.882
C00824=1099.972,35.560,-55.278,176.410,14.792,151.883
C00825=1099.966,35.311,-55.262,176.408,14.792,151.883
C00826=1099.961,35.061,-55.247,176.405,14.792,151.884
C00827=1099.955,34.812,-55.232,176.402,14.791,151.884
C00828=1099.949,34.562,-55.217,176.400,14.790,151.884
C00829=1099.943,34.313,-55.202,176.398,14.790,151.885
C00830=1099.938,34.063,-55.186,176.396,14.790,151.885
C00831=1099.932,33.814,-55.172,176.393,14.789,151.886
C00832=1099.926,33.564,-55.156,176.391,14.788,151.886
C00833=1099.920,33.315,-55.142,176.389,14.788,151.886
C00834=1099.914,33.065,-55.125,176.387,14.787,151.887
C00835=1099.908,32.816,-55.111,176.384,14.786,151.887
C00836=1099.903,32.567,-55.095,176.382,14.786,151.888
C00837=1099.897,32.317,-55.080,176.380,14.785,151.888
C00838=1099.891,32.044,-55.064,176.377,14.784,151.888
C00839=1099.885,31.770,-55.048,176.375,14.784,151.889
C00840=1099.879,31.498,-55.031,176.372,14.783,151.889
C00841=1099.872,31.225,-55.015,176.370,14.783,151.890
C00842=1099.867,30.975,-54.999,176.367,14.783,151.890
C00843=1099.861,30.726,-54.985,176.365,14.781,151.890
C00844=1099.855,30.476,-54.969,176.363,14.781,151.891
C00845=1099.850,30.227,-54.955,176.360,14.781,151.891
C00846=1099.844,29.977,-54.939,176.358,14.779,151.892
C00847=1099.838,29.728,-54.924,176.356,14.779,151.892
C00848=1099.832,29.478,-54.909,176.353,14.779,151.892
C00849=1099.827,29.229,-54.894,176.351,14.778,151.893
C00850=1099.821,28.979,-54.879,176.348,14.777,151.893
C00851=1099.815,28.730,-54.864,176.346,14.777,151.893
C00852=1099.810,28.480,-54.849,176.344,14.776,151.894
C00853=1099.804,28.231,-54.834,176.342,14.776,151.894
C00854=1099.798,27.981,-54.820,176.339,14.775,151.895
C00855=1099.793,27.732,-54.805,176.337,14.774,151.895
C00856=1099.786,27.482,-54.790,176.335,14.774,151.895
C00857=1099.781,27.233,-54.775,176.333,14.773,151.896
C00858=1099.775,26.983,-54.760,176.330,14.772,151.896
C00859=1099.769,26.734,-54.745,176.328,14.772,151.896
C00860=1099.763,26.484,-54.729,176.326,14.771,151.897
C00861=1099.758,26.235,-54.715,176.324,14.771,151.897
C00862=1099.752,25.985,-54.701,176.321,14.770,151.898
C00863=1099.747,25.736,-54.685,176.319,14.769,151.898
C00864=1099.740,25.486,-54.671,176.317,14.769,151.898
C00865=1099.734,25.237,-54.656,176.315,14.768,151.899
C00866=1099.728,24.987,-54.641,176.312,14.767,151.899
C00867=1099.723,24.737,-54.627,176.310,14.767,151.899
C00868=1099.717,24.488,-54.612,176.308,14.766,151.900
C00869=1099.711,24.239,-54.597,176.306,14.766,151.900
C00870=1099.706,23.989,-54.582,176.304,14.765,151.900
C00871=1099.700,23.740,-54.567,176.301,14.764,151.901
C00872=1099.694,23.490,-54.553,176.299,14.764,151.901
C00873=1099.689,23.240,-54.537,176.297,14.763,151.902
C00874=1099.683,22.991,-54.523,176.295,14.763,151.902
C00875=1099.677,22.741,-54.509,176.292,14.762,151.902
C00876=1099.671,22.492,-54.494,176.290,14.761,151.903
C00877=1099.666,22.243,-54.479,176.288,14.761,151.903
C00878=1099.660,21.993,-54.464,176.286,14.760,151.903
C00879=1099.654,21.744,-54.450,176.283,14.759,151.904
C00880=1099.648,21.494,-54.435,176.281,14.759,151.904
C00881=1099.643,21.245,-54.420,176.279,14.758,151.904
C00882=1099.637,20.995,-54.406,176.277,14.758,151.905
C00883=1099.631,20.745,-54.391,176.274,14.756,151.905
C00884=1099.625,20.496,-54.377,176.272,14.756,151.905
C00885=1099.620,20.247,-54.362,176.270,14.756,151.906
C00886=1099.614,19.997,-54.347,176.268,14.755,151.906
C00887=1099.608,19.748,-54.333,176.266,14.754,151.907
C00888=1099.602,19.498,-54.318,176.263,14.753,151.907
C00889=1099.596,19.249,-54.304,176.261,14.753,151.907
C00890=1099.591,18.999,-54.290,176.259,14.752,151.907
C00891=1099.585,18.749,-54.274,176.257,14.752,151.908
C00892=1099.579,18.500,-54.260,176.254,14.750,151.908
C00893=1099.573,18.250,-54.246,176.252,14.750,151.909
C00894=1099.567,18.001,-54.231,176.250,14.749,151.909
C00895=1099.562,17.751,-54.217,176.248,14.749,151.909
C00896=1099.556,17.502,-54.202,176.246,14.748,151.910
C00897=1099.550,17.252,-54.188,176.243,14.747,151.910
C00898=1099.545,17.003,-54.173,176.241,14.747,151.910
C00899=1099.539,16.753,-54.158,176.239,14.746,151.911
C00900=1099.533,16.504,-54.144,176.237,14.746,151.911
C00901=1099.527,16.255,-54.130,176.235,14.745,151.911
C00902=1099.521,15.983,-54.115,176.232,14.744,151.912
C00903=1099.515,15.711,-54.099,176.230,14.744,151.912
C00904=1099.508,15.440,-54.083,176.227,14.743,151.912
C00905=1099.502,15.167,-54.067,176.225,14.742,151.913
C00906=1099.497,14.918,-54.053,176.223,14.742,151.913
C00907=1099.491,14.669,-54.039,176.221,14.741,151.913
C00908=1099.485,14.419,-54.024,176.218,14.740,151.914
C00909=1099.479,14.169,-54.010,176.216,14.739,151.914
C00910=1099.473,13.921,-53.995,176.214,14.739,151.915
C00911=1099.467,13.670,-53.981,176.212,14.738,151.915
C00912=1099.462,13.421,-53.967,176.210,14.738,151.915
C00913=1099.456,13.172,-53.953,176.207,14.736,151.916
C00914=1099.450,12.921,-53.939,176.205,14.736,151.916
C00915=1099.444,12.672,-53.924,176.203,14.735,151.916
C00916=1099.439,12.423,-53.910,176.201,14.735,151.917
C00917=1099.432,12.173,-53.895,176.199,14.734,151.917
C00918=1099.427,11.924,-53.881,176.196,14.733,151.917
C00919=1099.421,11.674,-53.867,176.194,14.733,151.918
C00920=1099.414,11.425,-53.853,176.193,14.732,151.918
C00921=1099.409,11.175,-53.839,176.190,14.732,151.918
C00922=1099.403,10.926,-53.825,176.189,14.731,151.919
C00923=1099.397,10.676,-53.810,176.186,14.730,151.919
C00924=1099.392,10.426,-53.797,176.184,14.729,151.919
C00925=1099.386,10.177,-53.783,176.181,14.729,151.920
C00926=1099.380,9.927,-53.768,176.180,14.728,151.920
C00927=1099.374,9.678,-53.754,176.177,14.728,151.920
C00928=1099.369,9.428,-53.740,176.176,14.727,151.921
C00929=1099.363,9.179,-53.725,176.173,14.726,151.921
C00930=1099.356,8.929,-53.712,176.171,14.725,151.921
C00931=1099.351,8.679,-53.698,176.169,14.725,151.922
C00932=1099.345,8.431,-53.683,176.167,14.724,151.922
C00933=1099.339,8.181,-53.669,176.165,14.724,151.922
C00934=1099.333,7.931,-53.655,176.162,14.722,151.923
C00935=1099.328,7.681,-53.641,176.160,14.722,151.923
C00936=1099.322,7.432,-53.627,176.158,14.721,151.923
C00937=1099.316,7.183,-53.614,176.156,14.721,151.924
C00938=1099.310,6.933,-53.599,176.154,14.720,151.924
C00939=1099.304,6.683,-53.585,176.152,14.719,151.924
C00940=1099.298,6.434,-53.571,176.149,14.719,151.925
C00941=1099.293,6.185,-53.557,176.147,14.718,151.925
C00942=1099.288,5.935,-53.543,176.145,14.717,151.925
C00943=1099.281,5.685,-53.530,176.143,14.717,151.925
C00944=1099.275,5.435,-53.516,176.141,14.716,151.926
C00945=1099.269,5.186,-53.501,176.139,14.715,151.926
C00946=1099.264,4.937,-53.487,176.137,14.714,151.926
C00947=1099.258,4.687,-53.473,176.135,14.714,151.927
C00948=1099.252,4.437,-53.459,176.132,14.713,151.927
C00949=1099.246,4.188,-53.446,176.131,14.712,151.927
C00950=1099.241,3.938,-53.432,176.129,14.712,151.928
C00951=1099.235,3.689,-53.418,176.127,14.711,151.928
C00952=1099.229,3.440,-53.404,176.124,14.710,151.928
C00953=1099.224,3.190,-53.390,176.122,14.709,151.929
C00954=1099.217,2.940,-53.376,176.120,14.709,151.929
C00955=1099.212,2.691,-53.362,176.118,14.708,151.929
C00956=1099.206,2.441,-53.348,176.116,14.707,151.930
C00957=1099.201,2.191,-53.334,176.114,14.707,151.930
C00958=1099.195,1.942,-53.321,176.111,14.706,151.930
C00959=1099.189,1.693,-53.307,176.109,14.705,151.931
C00960=1099.184,1.443,-53.293,176.107,14.704,151.931
C00961=1099.178,1.193,-53.280,176.106,14.704,151.931
C00962=1099.172,0.943,-53.265,176.103,14.703,151.931
C00963=1099.166,0.694,-53.252,176.102,14.703,151.932
C00964=1099.160,0.444,-53.238,176.099,14.701,151.932
C00965=1099.155,0.195,-53.224,176.097,14.701,151.932
C00966=1099.148,-0.074,-53.209,176.095,14.700,151.933
C00967=1099.143,-0.344,-53.194,176.093,14.699,151.933
C00968=1099.136,-0.614,-53.180,176.090,14.698,151.933
C00969=1099.130,-0.884,-53.166,176.088,14.698,151.934
C00970=1099.124,-1.133,-53.152,176.086,14.697,151.934
C00971=1099.118,-1.384,-53.138,176.084,14.696,151.934
C00972=1099.113,-1.633,-53.124,176.082,14.696,151.935
C00973=1099.107,-1.882,-53.110,176.079,14.695,151.935
C00974=1099.101,-2.132,-53.097,176.078,14.694,151.935
C00975=1099.096,-2.382,-53.083,176.076,14.693,151.935
C00976=1099.090,-2.631,-53.069,176.074,14.693,151.936
C00977=1099.084,-2.880,-53.056,176.072,14.692,151.936
C00978=1099.079,-3.130,-53.042,176.070,14.691,151.936
C00979=1099.073,-3.380,-53.028,176.068,14.690,151.937
C00980=1099.067,-3.629,-53.015,176.065,14.689,151.937
C00981=1099.061,-3.878,-53.001,176.063,14.689,151.937
C00982=1099.055,-4.128,-52.987,176.061,14.688,151.938
C00983=1099.050,-4.378,-52.974,176.059,14.687,151.938
C00984=1099.043,-4.628,-52.961,176.057,14.687,151.938
C00985=1099.038,-4.877,-52.947,176.055,14.686,151.939
C00986=1099.032,-5.127,-52.933,176.053,14.685,151.939
C00987=1099.026,-5.376,-52.920,176.052,14.685,151.939
C00988=1099.020,-5.625,-52.906,176.049,14.684,151.939
C00989=1099.014,-5.875,-52.892,176.047,14.683,151.940
C00990=1099.008,-6.125,-52.880,176.045,14.682,151.940
C00991=1099.003,-6.375,-52.866,176.043,14.682,151.940
C00992=1098.997,-6.624,-52.853,176.041,14.681,151.941
C00993=1098.991,-6.873,-52.839,176.039,14.681,151.941
C00994=1098.985,-7.123,-52.826,176.037,14.680,151.941
C00995=1098.980,-7.372,-52.812,176.035,14.679,151.941
C00996=1098.974,-7.622,-52.799,176.032,14.678,151.942
C00997=1098.968,-7.872,-52.785,176.030,14.677,151.942
C00998=1098.961,-8.122,-52.772,176.028,14.677,151.942
C00999=1098.956,-8.371,-52.758,176.027,14.676,151.943
C01000=1098.950,-8.621,-52.745,176.024,14.676,151.943
C01001=1098.944,-8.870,-52.732,176.022,14.675,151.943
C01002=1098.938,-9.120,-52.718,176.021,14.674,151.944
C01003=1098.932,-9.369,-52.705,176.019,14.673,151.944
C01004=1098.927,-9.619,-52.692,176.017,14.673,151.944
C01005=1098.921,-9.869,-52.679,176.014,14.672,151.945
C01006=1098.915,-10.118,-52.665,176.012,14.671,151.945
C01007=1098.909,-10.367,-52.651,176.010,14.670,151.945
C01008=1098.904,-10.618,-52.638,176.008,14.669,151.945
C01009=1098.898,-10.867,-52.625,176.006,14.669,151.946
C01010=1098.891,-11.116,-52.612,176.004,14.668,151.946
C01011=1098.886,-11.366,-52.599,176.002,14.668,151.946
C01012=1098.880,-11.616,-52.585,176.000,14.667,151.947
C01013=1098.875,-11.865,-52.571,175.999,14.666,151.947
C01014=1098.869,-12.115,-52.559,175.997,14.665,151.947
C01015=1098.862,-12.364,-52.546,175.994,14.664,151.948
C01016=1098.857,-12.614,-52.532,175.992,14.664,151.948
C01017=1098.852,-12.863,-52.520,175.990,14.663,151.948
C01018=1098.846,-13.113,-52.506,175.988,14.662,151.948
C01019=1098.840,-13.363,-52.493,175.986,14.661,151.949
C01020=1098.834,-13.612,-52.480,175.984,14.661,151.949
C01021=1098.829,-13.861,-52.466,175.982,14.660,151.949
C01022=1098.823,-14.111,-52.453,175.980,14.660,151.950
C01023=1098.817,-14.361,-52.440,175.978,14.659,151.950
C01024=1098.811,-14.611,-52.427,175.977,14.658,151.950
C01025=1098.805,-14.860,-52.414,175.975,14.657,151.950
C01026=1098.800,-15.110,-52.401,175.972,14.656,151.951
C01027=1098.794,-15.359,-52.387,175.970,14.655,151.951
C01028=1098.788,-15.609,-52.374,175.968,14.655,151.951
C01029=1098.782,-15.859,-52.361,175.966,14.654,151.952
C01030=1098.776,-16.127,-52.347,175.964,14.653,151.952
C01031=1098.769,-16.394,-52.333,175.962,14.653,151.952
C01032=1098.763,-16.663,-52.320,175.959,14.652,151.953
C01033=1098.757,-16.931,-52.305,175.957,14.651,151.953
C01034=1098.751,-17.181,-52.292,175.956,14.650,151.953
C01035=1098.745,-17.430,-52.279,175.954,14.650,151.953
C01036=1098.739,-17.680,-52.266,175.952,14.649,151.954
C01037=1098.733,-17.929,-52.254,175.950,14.649,151.954
C01038=1098.728,-18.178,-52.240,175.948,14.648,151.954
C01039=1098.722,-18.428,-52.227,175.946,14.647,151.954
C01040=1098.716,-18.678,-52.214,175.944,14.646,151.955
C01041=1098.710,-18.927,-52.201,175.942,14.646,151.955
C01042=1098.703,-19.177,-52.188,175.940,14.645,151.955
C01043=1098.698,-19.427,-52.175,175.938,14.644,151.956
C01044=1098.692,-19.677,-52.162,175.936,14.644,151.956
C01045=1098.686,-19.926,-52.149,175.934,14.642,151.956
C01046=1098.680,-20.176,-52.137,175.932,14.642,151.956
C01047=1098.674,-20.425,-52.123,175.930,14.641,151.957
C01048=1098.669,-20.674,-52.111,175.928,14.640,151.957
C01049=1098.663,-20.924,-52.097,175.926,14.639,151.957
C01050=1098.657,-21.174,-52.085,175.924,14.639,151.958
C01051=1098.651,-21.424,-52.072,175.922,14.638,151.958
C01052=1098.645,-21.673,-52.059,175.920,14.638,151.958
C01053=1098.639,-21.923,-52.046,175.918,14.637,151.958
C01054=1098.633,-22.173,-52.034,175.916,14.636,151.959
C01055=1098.627,-22.422,-52.021,175.914,14.635,151.959
C01056=1098.623,-22.672,-52.008,175.913,14.635,151.959
C01057=1098.617,-22.921,-51.995,175.911,14.634,151.960
C01058=1098.611,-23.171,-51.982,175.909,14.634,151.960
C01059=1098.605,-23.421,-51.969,175.907,14.633,151.960
C01060=1098.599,-23.670,-51.957,175.905,14.632,151.960
C01061=1098.592,-23.920,-51.944,175.903,14.631,151.961
C01062=1098.587,-24.169,-51.931,175.901,14.631,151.961
C01063=1098.581,-24.419,-51.919,175.898,14.629,151.961
C01064=1098.576,-24.668,-51.905,175.896,14.628,151.962
C01065=1098.570,-24.918,-51.892,175.895,14.628,151.962
C01066=1098.564,-25.168,-51.880,175.893,14.627,151.962
C01067=1098.559,-25.417,-51.868,175.891,14.626,151.962
C01068=1098.552,-25.667,-51.854,175.889,14.626,151.963
C01069=1098.547,-25.916,-51.842,175.887,14.625,151.963
C01070=1098.541,-26.166,-51.829,175.885,14.624,151.963
C01071=1098.535,-26.416,-51.817,175.883,14.624,151.964
C01072=1098.529,-26.665,-51.804,175.881,14.623,151.964
C01073=1098.523,-26.915,-51.791,175.879,14.622,151.964
C01074=1098.517,-27.165,-51.779,175.877,14.621,151.964
C01075=1098.511,-27.414,-51.766,175.876,14.621,151.965
C01076=1098.505,-27.664,-51.753,175.874,14.620,151.965
C01077=1098.500,-27.913,-51.741,175.872,14.619,151.965
C01078=1098.494,-28.163,-51.728,175.870,14.619,151.966
C01079=1098.488,-28.413,-51.716,175.868,14.618,151.966
C01080=1098.482,-28.663,-51.703,175.866,14.617,151.966
C01081=1098.476,-28.912,-51.690,175.864,14.617,151.966
C01082=1098.470,-29.162,-51.677,175.862,14.616,151.967
C01083=1098.465,-29.411,-51.665,175.860,14.615,151.967
C01084=1098.459,-29.661,-51.653,175.858,14.614,151.967
C01085=1098.453,-29.911,-51.640,175.856,14.614,151.967
C01086=1098.446,-30.160,-51.628,175.854,14.613,151.968
C01087=1098.440,-30.410,-51.615,175.852,14.613,151.968
C01088=1098.435,-30.659,-51.603,175.850,14.612,151.968
C01089=1098.429,-30.908,-51.590,175.849,14.611,151.969
C01090=1098.423,-31.158,-51.577,175.847,14.610,151.969
C01091=1098.417,-31.408,-51.565,175.845,14.610,151.969
C01092=1098.412,-31.657,-51.553,175.843,14.609,151.969
C01093=1098.406,-31.907,-51.540,175.841,14.608,151.970
C01094=1098.399,-32.174,-51.527,175.839,14.608,151.970
C01095=1098.393,-32.442,-51.513,175.836,14.606,151.970
C01096=1098.387,-32.710,-51.500,175.834,14.606,151.971
C01097=1098.380,-32.977,-51.487,175.833,14.605,151.971
C01098=1098.375,-33.226,-51.475,175.831,14.604,151.971
C01099=1098.369,-33.476,-51.462,175.829,14.603,151.971
C01100=1098.363,-33.726,-51.450,175.827,14.603,151.972
C01101=1098.357,-33.975,-51.437,175.825,14.602,151.972
C01102=1098.352,-34.225,-51.425,175.823,14.601,151.972
C01103=1098.346,-34.474,-51.413,175.821,14.601,151.973
C01104=1098.339,-34.724,-51.401,175.819,14.600,151.973
C01105=1098.334,-34.973,-51.388,175.817,14.599,151.973
C01106=1098.328,-35.223,-51.376,175.815,14.599,151.973
C01107=1098.322,-35.473,-51.363,175.813,14.598,151.974
C01108=1098.317,-35.722,-51.351,175.812,14.597,151.974
C01109=1098.311,-35.972,-51.339,175.810,14.596,151.974
C01110=1098.304,-36.222,-51.327,175.808,14.596,151.974
C01111=1098.298,-36.472,-51.314,175.806,14.595,151.975
C01112=1098.293,-36.721,-51.302,175.804,14.594,151.975
C01113=1098.287,-36.971,-51.289,175.802,14.593,151.975
C01114=1098.281,-37.220,-51.277,175.800,14.593,151.975
C01115=1098.275,-37.469,-51.265,175.798,14.592,151.976
C01116=1098.269,-37.719,-51.253,175.797,14.591,151.976
C01117=1098.263,-37.969,-51.240,175.795,14.590,151.976
C01118=1098.258,-38.218,-51.228,175.793,14.590,151.976
C01119=1098.252,-38.468,-51.215,175.791,14.589,151.977
C01120=1098.246,-38.718,-51.204,175.789,14.589,151.977
C01121=1098.240,-38.968,-51.192,175.787,14.588,151.977
C01122=1098.234,-39.217,-51.179,175.785,14.587,151.978
C01123=1098.228,-39.467,-51.167,175.783,14.586,151.978
C01124=1098.222,-39.716,-51.155,175.781,14.586,151.978
C01125=1098.216,-39.966,-51.143,175.780,14.586,151.978
C01126=1098.210,-40.216,-51.131,175.778,14.585,151.979
C01127=1098.205,-40.465,-51.118,175.776,14.584,151.979
C01128=1098.199,-40.715,-51.107,175.774,14.583,151.979
C01129=1098.192,-40.965,-51.095,175.773,14.583,151.979
C01130=1098.187,-41.214,-51.082,175.770,14.582,151.980
C01131=1098.181,-41.464,-51.070,175.769,14.582,151.980
C01132=1098.174,-41.714,-51.058,175.767,14.581,151.980
C01133=1098.169,-41.963,-51.046,175.765,14.580,151.981
C01134=1098.163,-42.213,-51.034,175.763,14.579,151.981
C01135=1098.157,-42.463,-51.022,175.761,14.579,151.981
C01136=1098.152,-42.712,-51.010,175.759,14.578,151.981
C01137=1098.145,-42.962,-50.998,175.757,14.577,151.982
C01138=1098.139,-43.211,-50.985,175.755,14.576,151.982
C01139=1098.133,-43.461,-50.974,175.754,14.576,151.982
C01140=1098.127,-43.711,-50.962,175.752,14.575,151.983
C01141=1098.122,-43.960,-50.950,175.749,14.575,151.983
C01142=1098.115,-44.210,-50.938,175.748,14.574,151.983
C01143=1098.110,-44.460,-50.926,175.746,14.573,151.983
C01144=1098.104,-44.709,-50.914,175.744,14.572,151.984
C01145=1098.098,-44.959,-50.902,175.742,14.572,151.984
C01146=1098.093,-45.208,-50.889,175.741,14.572,151.984
C01147=1098.086,-45.458,-50.878,175.739,14.571,151.984
C01148=1098.080,-45.708,-50.866,175.737,14.570,151.985
C01149=1098.074,-45.957,-50.854,175.735,14.569,151.985
C01150=1098.069,-46.207,-50.842,175.733,14.569,151.985
C01151=1098.063,-46.456,-50.831,175.731,14.568,151.986
C01152=1098.057,-46.706,-50.818,175.730,14.567,151.986
C01153=1098.051,-46.957,-50.806,175.728,14.566,151.986
C01154=1098.045,-47.206,-50.795,175.726,14.566,151.986
C01155=1098.039,-47.455,-50.782,175.724,14.565,151.987
C01156=1098.033,-47.705,-50.771,175.722,14.565,151.987
C01157=1098.027,-47.955,-50.759,175.720,14.564,151.987
C01158=1098.021,-48.222,-50.746,175.718,14.563,151.988
C01159=1098.015,-48.490,-50.733,175.716,14.562,151.988
C01160=1098.008,-48.758,-50.721,175.714,14.562,151.988
C01161=1098.002,-49.025,-50.709,175.712,14.561,151.988
C01162=1097.996,-49.275,-50.696,175.710,14.560,151.989
C01163=1097.990,-49.524,-50.685,175.709,14.559,151.989
C01164=1097.985,-49.774,-50.673,175.707,14.559,151.989
C01165=1097.978,-50.024,-50.661,175.705,14.558,151.989
C01166=1097.973,-50.274,-50.649,175.703,14.557,151.990
C01167=1097.967,-50.523,-50.637,175.702,14.557,151.990
C01168=1097.961,-50.772,-50.625,175.700,14.557,151.990
C01169=1097.955,-51.022,-50.614,175.698,14.556,151.991
C01170=1097.949,-51.271,-50.602,175.696,14.555,151.991
C01171=1097.943,-51.522,-50.591,175.694,14.554,151.991
C01172=1097.937,-51.771,-50.579,175.692,14.554,151.991
C01173=1097.931,-52.021,-50.568,175.690,14.553,151.992
C01174=1097.925,-52.271,-50.555,175.688,14.552,151.992
C01175=1097.919,-52.520,-50.544,175.686,14.552,151.992
C01176=1097.913,-52.770,-50.532,175.684,14.551,151.993
C01177=1097.906,-53.019,-50.521,175.683,14.551,151.993
C01178=1097.901,-53.269,-50.509,175.681,14.550,151.993
C01179=1097.894,-53.519,-50.497,175.679,14.550,151.993
C01180=1097.889,-53.768,-50.486,175.678,14.549,151.994
C01181=1097.883,-54.018,-50.473,175.676,14.548,151.994
C01182=1097.877,-54.268,-50.463,175.673,14.548,151.994
C01183=1097.870,-54.517,-50.451,175.672,14.547,151.995
C01184=1097.864,-54.767,-50.440,175.670,14.546,151.995
C01185=1097.859,-55.017,-50.427,175.668,14.546,151.995
C01186=1097.853,-55.266,-50.416,175.667,14.546,151.995
C01187=1097.846,-55.516,-50.404,175.665,14.545,151.996
C01188=1097.840,-55.766,-50.393,175.663,14.544,151.996
C01189=1097.835,-56.016,-50.382,175.661,14.543,151.996
C01190=1097.828,-56.265,-50.370,175.659,14.543,151.996
C01191=1097.822,-56.515,-50.359,175.657,14.542,151.997
C01192=1097.816,-56.764,-50.347,175.655,14.542,151.997
C01193=1097.811,-57.014,-50.335,175.653,14.541,151.997
C01194=1097.804,-57.264,-50.323,175.652,14.541,151.998
C01195=1097.798,-57.513,-50.313,175.650,14.540,151.998
C01196=1097.792,-57.763,-50.301,175.648,14.539,151.998
C01197=1097.787,-58.013,-50.289,175.647,14.538,151.998
C01198=1097.780,-58.263,-50.278,175.644,14.538,151.999
C01199=1097.774,-58.512,-50.266,175.642,14.537,151.999
C01200=1097.768,-58.762,-50.255,175.641,14.537,151.999
C01201=1097.762,-59.011,-50.244,175.639,14.536,152.000
C01202=1097.756,-59.261,-50.232,175.638,14.536,152.000
C01203=1097.751,-59.511,-50.221,175.636,14.535,152.000
C01204=1097.745,-59.760,-50.210,175.634,14.534,152.000
C01205=1097.738,-60.010,-50.198,175.632,14.534,152.001
C01206=1097.733,-60.259,-50.187,175.630,14.533,152.001
C01207=1097.727,-60.510,-50.175,175.628,14.533,152.001
C01208=1097.721,-60.759,-50.164,175.626,14.532,152.002
C01209=1097.715,-61.009,-50.152,175.625,14.532,152.002
C01210=1097.709,-61.258,-50.141,175.623,14.531,152.002
C01211=1097.702,-61.508,-50.129,175.621,14.530,152.002
C01212=1097.697,-61.758,-50.118,175.619,14.530,152.003
C01213=1097.691,-62.007,-50.107,175.617,14.529,152.003
C01214=1097.685,-62.257,-50.096,175.616,14.528,152.003
C01215=1097.679,-62.506,-50.084,175.614,14.528,152.003
C01216=1097.673,-62.756,-50.073,175.612,14.528,152.004
C01217=1097.667,-63.006,-50.062,175.610,14.527,152.004
C01218=1097.661,-63.256,-50.050,175.608,14.526,152.004
C01219=1097.655,-63.505,-50.039,175.607,14.525,152.004
C01220=1097.650,-63.755,-50.028,175.605,14.525,152.005
C01221=1097.643,-64.005,-50.017,175.604,14.525,152.005
C01222=1097.637,-64.273,-50.005,175.602,14.524,152.005
C01223=1097.631,-64.542,-49.992,175.599,14.524,152.006
C01224=1097.624,-64.811,-49.980,175.598,14.523,152.006
C01225=1097.618,-65.080,-49.968,175.596,14.522,152.006
C01226=1097.612,-65.330,-49.957,175.594,14.521,152.006
C01227=1097.606,-65.580,-49.946,175.592,14.521,152.007
C01228=1097.600,-65.830,-49.935,175.590,14.520,152.007
C01229=1097.594,-66.079,-49.924,175.588,14.519,152.007
C01230=1097.588,-66.328,-49.912,175.586,14.518,152.008
C01231=1097.582,-66.578,-49.901,175.585,14.519,152.008
C01232=1097.576,-66.828,-49.890,175.583,14.518,152.008
C01233=1097.571,-67.078,-49.878,175.581,14.517,152.008
C01234=1097.565,-67.328,-49.867,175.579,14.517,152.009
C01235=1097.559,-67.577,-49.856,175.577,14.516,152.009
C01236=1097.553,-67.826,-49.845,175.576,14.516,152.009
C01237=1097.547,-68.076,-49.833,175.574,14.515,152.009
C01238=1097.541,-68.326,-49.823,175.573,14.514,152.010
C01239=1097.535,-68.575,-49.812,175.571,14.513,152.010
C01240=1097.529,-68.826,-49.800,175.569,14.513,152.010
C01241=1097.523,-69.075,-49.790,175.567,14.512,152.011
C01242=1097.517,-69.325,-49.779,175.565,14.512,152.011
C01243=1097.511,-69.575,-49.767,175.564,14.512,152.011
C01244=1097.506,-69.825,-49.756,175.562,14.511,152.011
C01245=1097.500,-70.074,-49.745,175.560,14.510,152.012
C01246=1097.494,-70.324,-49.734,175.558,14.509,152.012
C01247=1097.488,-70.574,-49.723,175.557,14.509,152.012
C01248=1097.482,-70.823,-49.711,175.555,14.509,152.012
C01249=1097.476,-71.072,-49.701,175.553,14.508,152.013
C01250=1097.470,-71.322,-49.689,175.551,14.507,152.013
C01251=1097.464,-71.572,-49.678,175.549,14.507,152.013
C01252=1097.458,-71.821,-49.668,175.548,14.507,152.014
C01253=1097.452,-72.071,-49.656,175.546,14.506,152.014
C01254=1097.446,-72.321,-49.645,175.544,14.505,152.014
C01255=1097.441,-72.570,-49.635,175.542,14.504,152.014
C01256=1097.435,-72.820,-49.624,175.540,14.504,152.015
C01257=1097.429,-73.070,-49.612,175.539,14.504,152.015
C01258=1097.423,-73.320,-49.602,175.537,14.503,152.015
C01259=1097.417,-73.569,-49.591,175.536,14.502,152.015
C01260=1097.411,-73.819,-49.580,175.534,14.501,152.016
C01261=1097.405,-74.069,-49.569,175.532,14.502,152.016
C01262=1097.399,-74.318,-49.558,175.530,14.501,152.016
C01263=1097.394,-74.568,-49.547,175.528,14.500,152.017
C01264=1097.388,-74.818,-49.537,175.527,14.500,152.017
C01265=1097.382,-75.068,-49.525,175.525,14.499,152.017
C01266=1097.376,-75.318,-49.515,175.524,14.499,152.017
C01267=1097.370,-75.567,-49.504,175.521,14.498,152.018
C01268=1097.363,-75.817,-49.493,175.519,14.498,152.018
C01269=1097.357,-76.066,-49.482,175.518,14.497,152.018
C01270=1097.352,-76.316,-49.471,175.517,14.497,152.019
C01271=1097.346,-76.565,-49.460,175.515,14.496,152.019
C01272=1097.340,-76.816,-49.449,175.513,14.495,152.019
C01273=1097.334,-77.065,-49.438,175.511,14.495,152.020
C01274=1097.328,-77.315,-49.427,175.509,14.495,152.020
C01275=1097.321,-77.564,-49.417,175.508,14.494,152.020
C01276=1097.315,-77.814,-49.406,175.506,14.493,152.020
C01277=1097.310,-78.064,-49.396,175.504,14.493,152.021
C01278=1097.304,-78.314,-49.385,175.503,14.493,152.021
C01279=1097.298,-78.564,-49.374,175.500,14.492,152.021
C01280=1097.291,-78.813,-49.363,175.499,14.492,152.022
C01281=1097.286,-79.062,-49.352,175.497,14.491,152.022
C01282=1097.280,-79.312,-49.342,175.496,14.491,152.022
C01283=1097.274,-79.562,-49.330,175.494,14.490,152.022
C01284=1097.268,-79.812,-49.320,175.492,14.490,152.023
C01285=1097.262,-80.062,-49.309,175.490,14.489,152.023
C01286=1097.255,-80.333,-49.298,175.488,14.488,152.023
C01287=1097.249,-80.603,-49.286,175.487,14.488,152.023
C01288=1097.242,-80.875,-49.275,175.484,14.488,152.024
C01289=1097.235,-81.146,-49.263,175.483,14.487,152.024
C01290=1097.230,-81.396,-49.252,175.481,14.486,152.024
C01291=1097.223,-81.645,-49.242,175.479,14.486,152.025
C01292=1097.217,-81.896,-49.231,175.477,14.486,152.025
C01293=1097.211,-82.145,-49.220,175.476,14.485,152.025
C01294=1097.205,-82.394,-49.210,175.474,14.485,152.026
C01295=1097.199,-82.644,-49.199,175.471,14.484,152.026
C01296=1097.192,-82.894,-49.189,175.470,14.484,152.026
C01297=1097.187,-83.144,-49.178,175.468,14.484,152.027
C01298=1097.181,-83.393,-49.167,175.467,14.483,152.027
C01299=1097.174,-83.642,-49.157,175.465,14.483,152.027
C01300=1097.168,-83.893,-49.146,175.463,14.482,152.027
C01301=1097.163,-84.143,-49.136,175.461,14.482,152.028
C01302=1097.156,-84.392,-49.126,175.459,14.481,152.028
C01303=1097.150,-84.641,-49.115,175.458,14.481,152.028
C01304=1097.144,-84.891,-49.105,175.456,14.481,152.029
C01305=1097.138,-85.141,-49.094,175.454,14.480,152.029
C01306=1097.132,-85.391,-49.083,175.453,14.480,152.029
C01307=1097.126,-85.640,-49.073,175.451,14.479,152.030
C01308=1097.120,-85.890,-49.063,175.449,14.479,152.030
C01309=1097.115,-86.140,-49.052,175.448,14.479,152.030
C01310=1097.107,-86.389,-49.041,175.446,14.478,152.030
C01311=1097.102,-86.640,-49.031,175.444,14.478,152.031
C01312=1097.096,-86.889,-49.021,175.442,14.477,152.031
C01313=1097.090,-87.138,-49.010,175.441,14.477,152.031
C01314=1097.084,-87.388,-49.000,175.439,14.476,152.032
C01315=1097.077,-87.638,-48.989,175.437,14.476,152.032
C01316=1097.072,-87.888,-48.978,175.436,14.476,152.032
C01317=1097.065,-88.138,-48.968,175.434,14.475,152.032
C01318=1097.060,-88.387,-48.958,175.432,14.475,152.033
C01319=1097.053,-88.637,-48.948,175.431,14.475,152.033
C01320=1097.048,-88.886,-48.937,175.429,14.474,152.033
C01321=1097.041,-89.137,-48.926,175.427,14.473,152.034
C01322=1097.035,-89.386,-48.916,175.425,14.473,152.034
C01323=1097.029,-89.636,-48.905,175.423,14.473,152.034
C01324=1097.023,-89.885,-48.895,175.422,14.472,152.035
C01325=1097.018,-90.135,-48.885,175.420,14.471,152.035
C01326=1097.011,-90.384,-48.875,175.418,14.472,152.035
C01327=1097.005,-90.635,-48.864,175.416,14.471,152.035
C01328=1096.999,-90.884,-48.854,175.415,14.470,152.036
C01329=1096.993,-91.134,-48.844,175.413,14.470,152.036
C01330=1096.987,-91.384,-48.833,175.411,14.470,152.036
C01331=1096.981,-91.633,-48.823,175.409,14.469,152.037
C01332=1096.975,-91.883,-48.812,175.408,14.469,152.037
C01333=1096.969,-92.132,-48.802,175.406,14.469,152.037
C01334=1096.964,-92.382,-48.792,175.404,14.468,152.038
C01335=1096.957,-92.632,-48.782,175.403,14.468,152.038
C01336=1096.951,-92.882,-48.771,175.401,14.467,152.038
C01337=1096.945,-93.132,-48.761,175.399,14.467,152.039
C01338=1096.939,-93.382,-48.751,175.398,14.467,152.039
C01339=1096.933,-93.631,-48.740,175.396,14.466,152.039
C01340=1096.927,-93.881,-48.730,175.394,14.465,152.039
C01341=1096.921,-94.130,-48.720,175.393,14.466,152.040
C01342=1096.915,-94.380,-48.710,175.391,14.465,152.040
C01343=1096.909,-94.629,-48.700,175.389,14.464,152.040
C01344=1096.903,-94.880,-48.689,175.387,14.465,152.041
C01345=1096.897,-95.129,-48.679,175.386,14.464,152.041
C01346=1096.892,-95.379,-48.669,175.384,14.463,152.041
C01347=1096.885,-95.629,-48.659,175.383,14.463,152.041
C01348=1096.879,-95.879,-48.648,175.380,14.463,152.042
C01349=1096.873,-96.129,-48.639,175.379,14.463,152.042
C01350=1096.866,-96.401,-48.627,175.377,14.462,152.042
C01351=1096.860,-96.675,-48.616,175.375,14.462,152.043
C01352=1096.854,-96.948,-48.604,175.373,14.461,152.043
C01353=1096.847,-97.222,-48.594,175.371,14.461,152.043
C01354=1096.841,-97.471,-48.583,175.370,14.461,152.044
C01355=1096.835,-97.721,-48.573,175.368,14.460,152.044
C01356=1096.829,-97.971,-48.564,175.366,14.460,152.044
C01357=1096.823,-98.220,-48.553,175.365,14.459,152.045
C01358=1096.817,-98.470,-48.543,175.363,14.459,152.045
C01359=1096.811,-98.720,-48.533,175.361,14.459,152.045
C01360=1096.805,-98.969,-48.523,175.360,14.458,152.046
C01361=1096.799,-99.220,-48.513,175.358,14.458,152.046
C01362=1096.792,-99.469,-48.502,175.356,14.458,152.046
C01363=1096.786,-99.719,-48.493,175.354,14.457,152.046
C01364=1096.780,-99.969,-48.483,175.352,14.457,152.047
C01365=1096.774,-100.218,-48.472,175.351,14.457,152.047
C01366=1096.768,-100.468,-48.463,175.349,14.456,152.047
C01367=1096.762,-100.718,-48.453,175.348,14.457,152.048
C01368=1096.756,-100.967,-48.442,175.346,14.456,152.048
C01369=1096.750,-101.217,-48.433,175.344,14.455,152.048
C01370=1096.744,-101.467,-48.423,175.343,14.456,152.049
C01371=1096.738,-101.717,-48.412,175.341,14.455,152.049
C01372=1096.732,-101.966,-48.403,175.340,14.455,152.049
C01373=1096.725,-102.216,-48.393,175.337,14.454,152.050
C01374=1096.719,-102.465,-48.383,175.335,14.454,152.050
C01375=1096.714,-102.715,-48.373,175.334,14.454,152.050
C01376=1096.707,-102.965,-48.363,175.332,14.453,152.051
C01377=1096.701,-103.214,-48.353,175.331,14.453,152.051
C01378=1096.695,-103.464,-48.343,175.329,14.453,152.051
C01379=1096.689,-103.714,-48.333,175.327,14.452,152.051
C01380=1096.683,-103.964,-48.324,175.326,14.453,152.052
C01381=1096.677,-104.213,-48.313,175.324,14.452,152.052
C01382=1096.670,-104.463,-48.304,175.323,14.452,152.052
C01383=1096.665,-104.713,-48.294,175.320,14.452,152.053
C01384=1096.658,-104.964,-48.284,175.318,14.451,152.053
C01385=1096.652,-105.213,-48.273,175.317,14.451,152.053
C01386=1096.646,-105.463,-48.264,175.315,14.450,152.054
C01387=1096.640,-105.713,-48.254,175.314,14.450,152.054
C01388=1096.634,-105.963,-48.244,175.312,14.450,152.054
C01389=1096.628,-106.212,-48.234,175.310,14.449,152.055
C01390=1096.621,-106.462,-48.224,175.308,14.450,152.055
C01391=1096.616,-106.711,-48.215,175.307,14.449,152.055
C01392=1096.610,-106.961,-48.205,175.306,14.449,152.056
C01393=1096.604,-107.211,-48.195,175.303,14.449,152.056
C01394=1096.598,-107.460,-48.185,175.302,14.449,152.056
C01395=1096.592,-107.710,-48.176,175.300,14.448,152.057
C01396=1096.585,-107.959,-48.166,175.298,14.448,152.057
C01397=1096.580,-108.209,-48.156,175.297,14.448,152.057
C01398=1096.574,-108.459,-48.146,175.295,14.447,152.058
C01399=1096.568,-108.709,-48.137,175.294,14.447,152.058
C01400=1096.561,-108.958,-48.126,175.291,14.447,152.058
C01401=1096.555,-109.208,-48.117,175.290,14.447,152.058
C01402=1096.549,-109.458,-48.107,175.288,14.447,152.059
C01403=1096.543,-109.708,-48.098,175.286,14.446,152.059
C01404=1096.536,-109.957,-48.088,175.285,14.446,152.060
C01405=1096.530,-110.207,-48.079,175.283,14.445,152.060
C01406=1096.524,-110.457,-48.069,175.282,14.446,152.060
C01407=1096.518,-110.706,-48.058,175.280,14.445,152.060
C01408=1096.512,-110.956,-48.049,175.278,14.445,152.061
C01409=1096.506,-111.206,-48.039,175.276,14.445,152.061
C01410=1096.500,-111.456,-48.029,175.275,14.445,152.062
C01411=1096.494,-111.706,-48.020,175.273,14.444,152.062
C01412=1096.487,-111.955,-48.010,175.271,14.444,152.062
C01413=1096.481,-112.205,-48.001,175.270,14.444,152.062
C01414=1096.475,-112.467,-47.990,175.267,14.444,152.063
C01415=1096.468,-112.729,-47.980,175.266,14.444,152.063
C01416=1096.462,-112.991,-47.971,175.264,14.443,152.064
C01417=1096.455,-113.254,-47.960,175.262,14.443,152.064
C01418=1096.449,-113.504,-47.951,175.261,14.443,152.064
C01419=1096.443,-113.753,-47.941,175.259,14.442,152.064
C01420=1096.437,-114.003,-47.932,175.258,14.443,152.065
C01421=1096.431,-114.253,-47.922,175.256,14.442,152.065
C01422=1096.425,-114.502,-47.913,175.254,14.442,152.066
C01423=1096.419,-114.752,-47.903,175.252,14.442,152.066
C01424=1096.413,-115.002,-47.894,175.251,14.442,152.066
C01425=1096.406,-115.252,-47.884,175.249,14.441,152.066
C01426=1096.400,-115.502,-47.874,175.248,14.442,152.067
C01427=1096.394,-115.751,-47.865,175.246,14.441,152.067
C01428=1096.388,-116.001,-47.855,175.244,14.441,152.068
C01429=1096.382,-116.251,-47.846,175.242,14.441,152.068
C01430=1096.376,-116.501,-47.836,175.241,14.441,152.068
C01431=1096.369,-116.751,-47.827,175.239,14.440,152.068
C01432=1096.363,-117.000,-47.817,175.238,14.441,152.069
C01433=1096.358,-117.249,-47.808,175.236,14.440,152.069
C01434=1096.351,-117.499,-47.798,175.234,14.440,152.070
C01435=1096.345,-117.749,-47.789,175.232,14.440,152.070
C01436=1096.339,-117.999,-47.779,175.230,14.439,152.070
C01437=1096.333,-118.249,-47.770,175.229,14.440,152.071
C01438=1096.327,-118.498,-47.760,175.227,14.439,152.071
C01439=1096.321,-118.748,-47.750,175.225,14.439,152.071
C01440=1096.314,-118.998,-47.741,175.224,14.439,152.072
C01441=1096.308,-119.248,-47.731,175.222,14.439,152.072
C01442=1096.302,-119.498,-47.722,175.220,14.438,152.072
C01443=1096.295,-119.747,-47.713,175.219,14.439,152.073
C01444=1096.290,-119.996,-47.704,175.217,14.438,152.073
C01445=1096.284,-120.247,-47.695,175.216,14.438,152.073
C01446=1096.278,-120.496,-47.685,175.213,14.438,152.074
C01447=1096.271,-120.746,-47.676,175.212,14.438,152.074
C01448=1096.265,-120.996,-47.666,175.210,14.438,152.074
C01449=1096.259,-121.246,-47.656,175.209,14.438,152.075
C01450=1096.253,-121.496,-47.647,175.207,14.437,152.075
C01451=1096.247,-121.745,-47.637,175.205,14.438,152.075
C01452=1096.240,-121.994,-47.629,175.204,14.438,152.076
C01453=1096.235,-122.245,-47.620,175.202,14.437,152.076
C01454=1096.228,-122.494,-47.610,175.201,14.437,152.076
C01455=1096.222,-122.744,-47.601,175.199,14.437,152.077
C01456=1096.216,-122.994,-47.591,175.197,14.437,152.077
C01457=1096.210,-123.244,-47.582,175.195,14.437,152.077
C01458=1096.204,-123.494,-47.572,175.194,14.437,152.078
C01459=1096.197,-123.742,-47.563,175.192,14.436,152.078
C01460=1096.192,-123.993,-47.554,175.191,14.437,152.078
C01461=1096.185,-124.243,-47.545,175.189,14.436,152.079
C01462=1096.179,-124.492,-47.535,175.187,14.436,152.079
C01463=1096.173,-124.742,-47.526,175.185,14.436,152.080
C01464=1096.167,-124.992,-47.516,175.184,14.436,152.080
C01465=1096.160,-125.242,-47.508,175.182,14.436,152.080
C01466=1096.155,-125.491,-47.499,175.180,14.436,152.081
C01467=1096.148,-125.741,-47.489,175.178,14.436,152.081
C01468=1096.142,-125.991,-47.480,175.177,14.436,152.081
C01469=1096.135,-126.240,-47.471,175.175,14.435,152.082
C01470=1096.130,-126.491,-47.462,175.174,14.436,152.082
C01471=1096.123,-126.740,-47.452,175.172,14.436,152.082
C01472=1096.117,-126.990,-47.443,175.170,14.435,152.083
C01473=1096.111,-127.239,-47.434,175.169,14.436,152.083
C01474=1096.104,-127.502,-47.424,175.167,14.435,152.083
C01475=1096.098,-127.765,-47.415,175.165,14.436,152.084
C01476=1096.092,-128.027,-47.405,175.163,14.435,152.084
C01477=1096.090,-128.290,-47.394,175.162,14.434,152.084
C01478=1095.681,-128.311,-47.504,175.118,14.539,152.114
C01479=1095.682,-128.049,-47.515,175.119,14.540,152.114
C01480=1095.688,-127.787,-47.524,175.121,14.541,152.114
C01481=1095.695,-127.525,-47.534,175.123,14.541,152.114
C01482=1095.702,-127.263,-47.543,175.124,14.541,152.113
C01483=1095.707,-127.014,-47.552,175.126,14.542,152.113
C01484=1095.714,-126.764,-47.561,175.127,14.541,152.113
C01485=1095.720,-126.514,-47.571,175.129,14.541,152.112
C01486=1095.726,-126.264,-47.580,175.131,14.542,152.112
C01487=1095.732,-126.014,-47.589,175.132,14.541,152.112
C01488=1095.739,-125.765,-47.598,175.134,14.542,152.111
C01489=1095.745,-125.515,-47.608,175.136,14.542,152.111
C01490=1095.751,-125.266,-47.617,175.138,14.542,152.110
C01491=1095.757,-125.015,-47.626,175.139,14.542,152.110
C01492=1095.764,-124.766,-47.635,175.141,14.542,152.110
C01493=1095.770,-124.516,-47.645,175.142,14.542,152.110
C01494=1095.776,-124.266,-47.654,175.144,14.542,152.109
C01495=1095.782,-124.016,-47.664,175.146,14.542,152.109
C01496=1095.788,-123.767,-47.672,175.148,14.543,152.108
C01497=1095.794,-123.517,-47.682,175.149,14.542,152.108
C01498=1095.801,-123.267,-47.691,175.151,14.543,152.108
C01499=1095.807,-123.018,-47.700,175.152,14.543,152.107
C01500=1095.813,-122.768,-47.710,175.154,14.543,152.107
C01501=1095.819,-122.518,-47.719,175.156,14.543,152.107
C01502=1095.825,-122.268,-47.728,175.158,14.544,152.106
C01503=1095.831,-122.019,-47.737,175.159,14.543,152.106
C01504=1095.837,-121.769,-47.747,175.161,14.544,152.106
C01505=1095.844,-121.519,-47.756,175.162,14.544,152.105
C01506=1095.850,-121.269,-47.766,175.165,14.544,152.105
C01507=1095.856,-121.020,-47.775,175.166,14.544,152.105
C01508=1095.862,-120.770,-47.785,175.168,14.544,152.104
C01509=1095.868,-120.520,-47.794,175.169,14.544,152.104
C01510=1095.874,-120.270,-47.803,175.171,14.545,152.104
C01511=1095.880,-120.021,-47.812,175.172,14.545,152.103
C01512=1095.886,-119.771,-47.822,175.175,14.545,152.103
C01513=1095.892,-119.521,-47.831,175.176,14.545,152.103
C01514=1095.899,-119.271,-47.840,175.178,14.545,152.102
C01515=1095.905,-119.022,-47.850,175.179,14.545,152.102
C01516=1095.911,-118.772,-47.860,175.181,14.546,152.102
C01517=1095.918,-118.522,-47.869,175.182,14.546,152.101
C01518=1095.924,-118.272,-47.879,175.185,14.546,152.101
C01519=1095.930,-118.022,-47.888,175.186,14.546,152.101
C01520=1095.936,-117.773,-47.898,175.188,14.546,152.100
C01521=1095.942,-117.524,-47.907,175.189,14.546,152.100
C01522=1095.948,-117.274,-47.917,175.191,14.547,152.100
C01523=1095.954,-117.024,-47.926,175.192,14.547,152.099
C01524=1095.960,-116.774,-47.936,175.194,14.547,152.099
C01525=1095.966,-116.524,-47.945,175.196,14.547,152.099
C01526=1095.972,-116.275,-47.955,175.198,14.547,152.098
C01527=1095.979,-116.025,-47.964,175.199,14.547,152.098
C01528=1095.985,-115.775,-47.974,175.201,14.548,152.098
C01529=1095.991,-115.525,-47.984,175.203,14.548,152.097
C01530=1095.997,-115.275,-47.993,175.204,14.548,152.097
C01531=1096.003,-115.026,-48.003,175.206,14.549,152.097
C01532=1096.010,-114.776,-48.012,175.208,14.548,152.096
C01533=1096.016,-114.526,-48.022,175.210,14.549,152.096
C01534=1096.022,-114.276,-48.031,175.211,14.549,152.096
C01535=1096.027,-114.027,-48.041,175.213,14.549,152.095
C01536=1096.034,-113.777,-48.050,175.214,14.549,152.095
C01537=1096.040,-113.528,-48.060,175.216,14.550,152.095
C01538=1096.046,-113.278,-48.069,175.217,14.550,152.095
C01539=1096.053,-113.015,-48.079,175.220,14.550,152.094
C01540=1096.059,-112.751,-48.089,175.221,14.551,152.094
C01541=1096.065,-112.489,-48.099,175.223,14.550,152.093
C01542=1096.072,-112.226,-48.110,175.225,14.551,152.093
C01543=1096.078,-111.976,-48.119,175.226,14.551,152.093
C01544=1096.084,-111.726,-48.129,175.228,14.551,152.093
C01545=1096.090,-111.477,-48.138,175.230,14.552,152.092
C01546=1096.097,-111.227,-48.148,175.231,14.552,152.092
C01547=1096.103,-110.977,-48.158,175.233,14.553,152.092
C01548=1096.108,-110.727,-48.168,175.235,14.552,152.091
C01549=1096.114,-110.477,-48.177,175.237,14.553,152.091
C01550=1096.121,-110.227,-48.187,175.238,14.552,152.091
C01551=1096.127,-109.978,-48.197,175.240,14.553,152.090
C01552=1096.133,-109.728,-48.207,175.242,14.553,152.090
C01553=1096.139,-109.478,-48.216,175.243,14.554,152.090
C01554=1096.146,-109.229,-48.226,175.245,14.554,152.089
C01555=1096.152,-108.979,-48.235,175.247,14.554,152.089
C01556=1096.158,-108.729,-48.245,175.248,14.555,152.089
C01557=1096.164,-108.479,-48.255,175.250,14.554,152.088
C01558=1096.170,-108.230,-48.265,175.252,14.555,152.088
C01559=1096.176,-107.980,-48.275,175.254,14.556,152.088
C01560=1096.182,-107.730,-48.285,175.255,14.555,152.087
C01561=1096.188,-107.480,-48.294,175.257,14.556,152.087
C01562=1096.194,-107.231,-48.304,175.258,14.556,152.087
C01563=1096.201,-106.981,-48.314,175.260,14.556,152.086
C01564=1096.206,-106.731,-48.324,175.261,14.556,152.086
C01565=1096.213,-106.481,-48.334,175.264,14.557,152.086
C01566=1096.219,-106.232,-48.343,175.265,14.557,152.086
C01567=1096.225,-105.982,-48.353,175.267,14.558,152.085
C01568=1096.231,-105.733,-48.363,175.269,14.558,152.085
C01569=1096.237,-105.483,-48.373,175.270,14.558,152.085
C01570=1096.243,-105.233,-48.383,175.272,14.559,152.084
C01571=1096.249,-104.983,-48.392,175.274,14.559,152.084
C01572=1096.256,-104.734,-48.403,175.275,14.559,152.084
C01573=1096.261,-104.484,-48.413,175.277,14.559,152.083
C01574=1096.267,-104.234,-48.422,175.278,14.559,152.083
C01575=1096.273,-103.984,-48.432,175.280,14.560,152.083
C01576=1096.280,-103.735,-48.442,175.283,14.560,152.082
C01577=1096.285,-103.485,-48.452,175.284,14.560,152.082
C01578=1096.291,-103.235,-48.462,175.285,14.561,152.082
C01579=1096.298,-102.985,-48.472,175.287,14.561,152.081
C01580=1096.304,-102.736,-48.482,175.289,14.561,152.081
C01581=1096.310,-102.486,-48.492,175.291,14.562,152.081
C01582=1096.316,-102.236,-48.502,175.292,14.562,152.081
C01583=1096.322,-101.987,-48.512,175.294,14.562,152.080
C01584=1096.328,-101.737,-48.521,175.296,14.563,152.080
C01585=1096.334,-101.487,-48.532,175.297,14.563,152.080
C01586=1096.340,-101.238,-48.542,175.299,14.564,152.079
C01587=1096.346,-100.988,-48.551,175.300,14.564,152.079
C01588=1096.352,-100.738,-48.562,175.303,14.564,152.079
C01589=1096.358,-100.489,-48.572,175.304,14.565,152.078
C01590=1096.365,-100.239,-48.581,175.306,14.565,152.078
C01591=1096.370,-99.989,-48.592,175.307,14.565,152.078
C01592=1096.377,-99.739,-48.602,175.310,14.566,152.077
C01593=1096.383,-99.489,-48.612,175.311,14.566,152.077
C01594=1096.389,-99.239,-48.621,175.313,14.567,152.077
C01595=1096.395,-98.990,-48.632,175.314,14.566,152.077
C01596=1096.401,-98.740,-48.642,175.316,14.567,152.076
C01597=1096.407,-98.490,-48.651,175.318,14.568,152.076
C01598=1096.413,-98.241,-48.662,175.319,14.567,152.076
C01599=1096.419,-97.991,-48.672,175.321,14.568,152.075
C01600=1096.426,-97.742,-48.682,175.323,14.569,152.075
C01601=1096.431,-97.492,-48.692,175.324,14.568,152.075
C01602=1096.437,-97.242,-48.702,175.326,14.569,152.074
C01603=1096.445,-96.969,-48.714,175.328,14.570,152.074
C01604=1096.451,-96.694,-48.725,175.329,14.570,152.074
C01605=1096.457,-96.421,-48.736,175.331,14.570,152.074
C01606=1096.464,-96.148,-48.747,175.333,14.571,152.073
C01607=1096.470,-95.898,-48.757,175.335,14.572,152.073
C01608=1096.476,-95.649,-48.768,175.337,14.571,152.073
C01609=1096.482,-95.399,-48.777,175.339,14.572,152.072
C01610=1096.488,-95.149,-48.788,175.340,14.573,152.072
C01611=1096.494,-94.900,-48.798,175.342,14.573,152.072
C01612=1096.499,-94.650,-48.809,175.344,14.573,152.071
C01613=1096.506,-94.400,-48.818,175.346,14.574,152.071
C01614=1096.512,-94.150,-48.829,175.347,14.574,152.071
C01615=1096.518,-93.900,-48.839,175.349,14.575,152.071
C01616=1096.524,-93.650,-48.849,175.351,14.575,152.070
C01617=1096.530,-93.401,-48.859,175.352,14.575,152.070
C01618=1096.535,-93.151,-48.870,175.354,14.576,152.070
C01619=1096.542,-92.902,-48.880,175.356,14.576,152.069
C01620=1096.548,-92.652,-48.891,175.357,14.576,152.069
C01621=1096.554,-92.402,-48.900,175.359,14.577,152.069
C01622=1096.560,-92.153,-48.911,175.361,14.577,152.069
C01623=1096.565,-91.903,-48.921,175.362,14.578,152.068
C01624=1096.572,-91.653,-48.932,175.364,14.578,152.068
C01625=1096.578,-91.403,-48.942,175.366,14.579,152.068
C01626=1096.584,-91.154,-48.952,175.368,14.579,152.067
C01627=1096.589,-90.904,-48.963,175.369,14.579,152.067
C01628=1096.596,-90.654,-48.973,175.371,14.580,152.067
C01629=1096.601,-90.404,-48.983,175.373,14.581,152.067
C01630=1096.608,-90.155,-48.993,175.374,14.580,152.066
C01631=1096.614,-89.905,-49.005,175.376,14.581,152.066
C01632=1096.620,-89.655,-49.014,175.378,14.582,152.066
C01633=1096.626,-89.406,-49.025,175.379,14.582,152.065
C01634=1096.632,-89.155,-49.035,175.381,14.583,152.065
C01635=1096.638,-88.906,-49.045,175.383,14.583,152.065
C01636=1096.644,-88.657,-49.056,175.384,14.583,152.065
C01637=1096.650,-88.407,-49.066,175.386,14.584,152.064
C01638=1096.656,-88.157,-49.077,175.388,14.585,152.064
C01639=1096.663,-87.908,-49.087,175.390,14.585,152.064
C01640=1096.668,-87.658,-49.098,175.391,14.585,152.063
C01641=1096.674,-87.408,-49.108,175.393,14.586,152.063
C01642=1096.680,-87.158,-49.118,175.395,14.586,152.063
C01643=1096.686,-86.908,-49.129,175.396,14.586,152.063
C01644=1096.693,-86.659,-49.140,175.398,14.587,152.062
C01645=1096.698,-86.409,-49.150,175.400,14.587,152.062
C01646=1096.704,-86.159,-49.161,175.402,14.588,152.062
C01647=1096.711,-85.910,-49.171,175.403,14.588,152.061
C01648=1096.717,-85.660,-49.182,175.405,14.589,152.061
C01649=1096.723,-85.410,-49.192,175.407,14.590,152.061
C01650=1096.729,-85.161,-49.203,175.409,14.589,152.060
C01651=1096.735,-84.911,-49.213,175.410,14.590,152.060
C01652=1096.741,-84.661,-49.223,175.412,14.591,152.060
C01653=1096.747,-84.411,-49.234,175.413,14.591,152.060
C01654=1096.754,-84.162,-49.244,175.415,14.592,152.059
C01655=1096.759,-83.913,-49.255,175.418,14.592,152.059
C01656=1096.765,-83.662,-49.266,175.419,14.593,152.059
C01657=1096.772,-83.413,-49.276,175.421,14.593,152.059
C01658=1096.778,-83.163,-49.287,175.422,14.594,152.058
C01659=1096.783,-82.914,-49.298,175.424,14.594,152.058
C01660=1096.789,-82.664,-49.308,175.427,14.594,152.058
C01661=1096.796,-82.414,-49.319,175.428,14.595,152.057
C01662=1096.801,-82.164,-49.330,175.429,14.595,152.057
C01663=1096.808,-81.915,-49.340,175.431,14.596,152.057
C01664=1096.813,-81.665,-49.350,175.432,14.596,152.057
C01665=1096.820,-81.415,-49.361,175.435,14.596,152.056
C01666=1096.826,-81.165,-49.372,175.437,14.597,152.056
C01667=1096.832,-80.894,-49.383,175.438,14.598,152.056
C01668=1096.839,-80.623,-49.394,175.440,14.599,152.055
C01669=1096.846,-80.351,-49.406,175.443,14.599,152.055
C01670=1096.852,-80.080,-49.418,175.444,14.599,152.055
C01671=1096.858,-79.831,-49.429,175.446,14.600,152.054
C01672=1096.864,-79.581,-49.439,175.447,14.600,152.054
C01673=1096.871,-79.331,-49.450,175.449,14.601,152.054
C01674=1096.876,-79.082,-49.461,175.451,14.602,152.054
C01675=1096.882,-78.832,-49.472,175.453,14.602,152.053
C01676=1096.888,-78.583,-49.483,175.454,14.602,152.053
C01677=1096.895,-78.332,-49.493,175.456,14.603,152.053
C01678=1096.900,-78.083,-49.504,175.458,14.604,152.052
C01679=1096.906,-77.833,-49.515,175.459,14.604,152.052
C01680=1096.912,-77.584,-49.525,175.461,14.605,152.052
C01681=1096.918,-77.334,-49.537,175.463,14.605,152.052
C01682=1096.924,-77.084,-49.548,175.465,14.606,152.051
C01683=1096.930,-76.835,-49.558,175.466,14.606,152.051
C01684=1096.937,-76.585,-49.569,175.468,14.606,152.051
C01685=1096.943,-76.335,-49.580,175.470,14.607,152.050
C01686=1096.948,-76.085,-49.590,175.472,14.608,152.050
C01687=1096.954,-75.836,-49.601,175.473,14.608,152.050
C01688=1096.960,-75.585,-49.612,175.475,14.609,152.050
C01689=1096.966,-75.336,-49.623,175.477,14.609,152.049
C01690=1096.972,-75.087,-49.633,175.479,14.610,152.049
C01691=1096.979,-74.837,-49.645,175.481,14.611,152.049
C01692=1096.984,-74.587,-49.655,175.482,14.611,152.049
C01693=1096.990,-74.338,-49.666,175.484,14.611,152.048
C01694=1096.996,-74.088,-49.677,175.486,14.612,152.048
C01695=1097.002,-73.838,-49.688,175.488,14.613,152.048
C01696=1097.008,-73.588,-49.699,175.490,14.613,152.047
C01697=1097.014,-73.339,-49.710,175.491,14.614,152.047
C01698=1097.019,-73.089,-49.721,175.493,14.614,152.047
C01699=1097.026,-72.839,-49.732,175.495,14.615,152.047
C01700=1097.032,-72.590,-49.743,175.496,14.616,152.046
C01701=1097.037,-72.340,-49.754,175.498,14.616,152.046
C01702=1097.043,-72.091,-49.765,175.499,14.617,152.046
C01703=1097.049,-71.841,-49.776,175.501,14.617,152.046
C01704=1097.055,-71.591,-49.787,175.503,14.618,152.045
C01705=1097.061,-71.342,-49.798,175.505,14.619,152.045
C01706=1097.067,-71.091,-49.809,175.507,14.620,152.045
C01707=1097.073,-70.842,-49.820,175.508,14.620,152.045
C01708=1097.079,-70.592,-49.831,175.510,14.620,152.044
C01709=1097.084,-70.343,-49.842,175.512,14.621,152.044
C01710=1097.090,-70.092,-49.854,175.514,14.622,152.044
C01711=1097.096,-69.843,-49.865,175.516,14.623,152.044
C01712=1097.101,-69.593,-49.875,175.517,14.623,152.043
C01713=1097.108,-69.343,-49.887,175.519,14.623,152.043
C01714=1097.114,-69.094,-49.898,175.520,14.624,152.043
C01715=1097.120,-68.845,-49.909,175.522,14.625,152.043
C01716=1097.126,-68.595,-49.920,175.524,14.626,152.042
C01717=1097.132,-68.345,-49.931,175.526,14.626,152.042
C01718=1097.137,-68.096,-49.942,175.527,14.626,152.042
C01719=1097.144,-67.846,-49.953,175.529,14.627,152.041
C01720=1097.149,-67.596,-49.964,175.531,14.627,152.041
C01721=1097.154,-67.346,-49.976,175.533,14.628,152.041
C01722=1097.161,-67.096,-49.987,175.535,14.629,152.041
C01723=1097.167,-66.847,-49.999,175.536,14.629,152.040
C01724=1097.173,-66.598,-50.009,175.538,14.630,152.040
C01725=1097.179,-66.347,-50.021,175.540,14.631,152.040
C01726=1097.185,-66.098,-50.032,175.542,14.631,152.040
C01727=1097.190,-65.849,-50.042,175.544,14.632,152.039
C01728=1097.197,-65.598,-50.054,175.546,14.633,152.039
C01729=1097.203,-65.349,-50.065,175.547,14.633,152.039
C01730=1097.208,-65.100,-50.077,175.548,14.634,152.039
C01731=1097.215,-64.831,-50.089,175.550,14.634,152.038
C01732=1097.221,-64.561,-50.100,175.552,14.635,152.038
C01733=1097.227,-64.292,-50.113,175.554,14.636,152.038
C01734=1097.234,-64.023,-50.125,175.556,14.636,152.037
C01735=1097.239,-63.773,-50.136,175.558,14.637,152.037
C01736=1097.245,-63.524,-50.147,175.560,14.637,152.037
C01737=1097.252,-63.274,-50.159,175.562,14.638,152.037
C01738=1097.258,-63.025,-50.170,175.564,14.639,152.036
C01739=1097.264,-62.774,-50.181,175.565,14.639,152.036
C01740=1097.270,-62.525,-50.192,175.567,14.640,152.036
C01741=1097.276,-62.275,-50.204,175.569,14.641,152.036
C01742=1097.281,-62.025,-50.216,175.571,14.641,152.035
C01743=1097.287,-61.776,-50.227,175.572,14.642,152.035
C01744=1097.294,-61.526,-50.239,175.574,14.643,152.035
C01745=1097.299,-61.277,-50.249,175.576,14.643,152.035
C01746=1097.306,-61.027,-50.261,175.577,14.644,152.034
C01747=1097.311,-60.777,-50.272,175.579,14.644,152.034
C01748=1097.317,-60.527,-50.284,175.581,14.645,152.034
C01749=1097.323,-60.278,-50.295,175.583,14.646,152.034
C01750=1097.329,-60.028,-50.306,175.585,14.647,152.033
C01751=1097.335,-59.779,-50.318,175.587,14.647,152.033
C01752=1097.341,-59.529,-50.329,175.589,14.648,152.033
C01753=1097.347,-59.279,-50.341,175.591,14.649,152.032
C01754=1097.353,-59.030,-50.352,175.592,14.649,152.032
C01755=1097.359,-58.780,-50.363,175.593,14.650,152.032
C01756=1097.365,-58.531,-50.375,175.596,14.650,152.032
C01757=1097.371,-58.280,-50.387,175.598,14.651,152.031
C01758=1097.377,-58.031,-50.398,175.599,14.651,152.031
C01759=1097.383,-57.781,-50.410,175.601,14.652,152.031
C01760=1097.389,-57.532,-50.421,175.603,14.653,152.030
C01761=1097.395,-57.282,-50.432,175.605,14.654,152.030
C01762=1097.401,-57.032,-50.444,175.606,14.654,152.030
C01763=1097.407,-56.782,-50.455,175.608,14.654,152.030
C01764=1097.413,-56.533,-50.467,175.610,14.655,152.029
C01765=1097.419,-56.283,-50.478,175.612,14.656,152.029
C01766=1097.425,-56.034,-50.490,175.614,14.657,152.029
C01767=1097.431,-55.784,-50.501,175.616,14.657,152.029
C01768=1097.437,-55.535,-50.513,175.617,14.658,152.028
C01769=1097.443,-55.285,-50.524,175.619,14.659,152.028
C01770=1097.448,-55.035,-50.536,175.620,14.659,152.028
C01771=1097.455,-54.785,-50.548,175.622,14.660,152.028
C01772=1097.461,-54.535,-50.559,175.624,14.660,152.027
C01773=1097.467,-54.286,-50.571,175.626,14.661,152.027
C01774=1097.473,-54.036,-50.582,175.628,14.661,152.027
C01775=1097.479,-53.787,-50.594,175.630,14.662,152.026
C01776=1097.485,-53.537,-50.605,175.632,14.663,152.026
C01777=1097.491,-53.288,-50.617,175.634,14.664,152.026
C01778=1097.497,-53.037,-50.629,175.636,14.664,152.026
C01779=1097.503,-52.789,-50.640,175.638,14.665,152.025
C01780=1097.509,-52.538,-50.652,175.639,14.665,152.025
C01781=1097.515,-52.288,-50.664,175.641,14.666,152.025
C01782=1097.521,-52.040,-50.676,175.643,14.667,152.025
C01783=1097.528,-51.789,-50.687,175.644,14.667,152.024
C01784=1097.533,-51.540,-50.699,175.646,14.668,152.024
C01785=1097.539,-51.290,-50.710,175.648,14.669,152.024
C01786=1097.546,-51.040,-50.722,175.650,14.670,152.024
C01787=1097.551,-50.791,-50.734,175.652,14.670,152.023
C01788=1097.558,-50.541,-50.746,175.654,14.671,152.023
C01789=1097.564,-50.292,-50.757,175.656,14.671,152.023
C01790=1097.569,-50.042,-50.769,175.658,14.672,152.022
C01791=1097.575,-49.793,-50.781,175.659,14.673,152.022
C01792=1097.581,-49.542,-50.793,175.661,14.673,152.022
C01793=1097.587,-49.293,-50.804,175.662,14.674,152.022
C01794=1097.593,-49.044,-50.817,175.664,14.675,152.022
C01795=1097.600,-48.776,-50.829,175.666,14.676,152.021
C01796=1097.605,-48.508,-50.842,175.668,14.676,152.021
C01797=1097.612,-48.240,-50.855,175.670,14.677,152.021
C01798=1097.618,-47.972,-50.868,175.673,14.678,152.020
C01799=1097.624,-47.722,-50.879,175.674,14.678,152.020
C01800=1097.630,-47.473,-50.891,175.676,14.679,152.020
C01801=1097.636,-47.223,-50.902,175.678,14.680,152.020
C01802=1097.641,-46.974,-50.915,175.680,14.680,152.019
C01803=1097.647,-46.724,-50.927,175.682,14.681,152.019
C01804=1097.653,-46.475,-50.939,175.683,14.682,152.019
C01805=1097.659,-46.224,-50.950,175.685,14.683,152.018
C01806=1097.665,-45.975,-50.962,175.687,14.683,152.018
C01807=1097.671,-45.726,-50.975,175.689,14.684,152.018
C01808=1097.677,-45.475,-50.986,175.691,14.685,152.018
C01809=1097.682,-45.226,-50.998,175.693,14.686,152.017
C01810=1097.688,-44.976,-51.011,175.695,14.686,152.017
C01811=1097.695,-44.726,-51.022,175.697,14.687,152.017
C01812=1097.700,-44.477,-51.034,175.698,14.688,152.017
C01813=1097.707,-44.227,-51.046,175.700,14.688,152.016
C01814=1097.712,-43.978,-51.058,175.702,14.689,152.016
